# B&R Automation Studio project NAEUL004C00R13L518F00 (part 66)

#### Act_Link.st
```iecst
(** 2021-08-01 **)
ACTION Act_Link:

	//Receive Alive Time
	p_tyParam.tRcvAlive	:= p_tyParam.tSndAlive * 2;

	//Board Depart
	bTransportFinish1 := p_bDSSMEMA1ConvStart AND EDGENEG(p_bPshrConvHvBrd);
	bTransportFinish2 := p_bDSSMEMA2ConvStart AND EDGENEG(p_bPshrConvHvBrd);
	bTransportFinish3 := p_bDSSMEMA3ConvStart AND EDGENEG(p_bPshrConvHvBrd);

	p_bDSHermesTransportFinished1:= bTransportFinish1 OR bTransportFinish2 OR bTransportFinish3;
	//Depart internal SMEMA
	IF EDGEPOS(p_bDSHermesTransportFinished1) THEN// p_bDSHermesTransportFinished1 OR p_bDSHermesTransportFinished2 OR p_bDSHermesTransportFinished3 ) THEN
		memset(ADR(p_bUSHermesARcvBoardInfo),0,SIZEOF(p_bUSHermesARcvBoardInfo));
		IF p_bLinkBrdAvlDataNewBrdAvl1stZ THEN //newly inserted
			//p_tyDSBoardDeparted1.tyData.sBoardId;
			IF NOT(p_bUSHermesARcvBoardInfo) THEN //create new BA
				fHermesGenerateUUID(ADR(tyDsInternalBoardDeparted.tyData.sBoardId) , p_tyDTStructure , pa_usiMacAddr);
				tyDsInternalBoardDeparted.tyData.sBoardIdCreatedBy := p_sMcId;
				tyDsInternalBoardDeparted.tyData.eFailedBoard  := BOOL_TO_USINT(p_bOpsTravLifGdBrdChk)*HermesGoodBoard + BOOL_TO_USINT(NOT(p_bOpsTravLifGdBrdChk))*HermesFailedBoard ;
				tyDsInternalBoardDeparted.tyData.sProductTypeId := p_tyProdRcpCurrRcp1.sRcpNm;
				tyDsInternalBoardDeparted.tyData.sTopBarcode := ''; //from UI
				tyDsInternalBoardDeparted.tyData.sBottomBarcode := ''; //from UI
				tyDsInternalBoardDeparted.tyData.rWidth := DINT_TO_REAL(p_tyProdRcpCurrRcp1.diWidthInUM)/1000;//Rcp
				tyDsInternalBoardDeparted.tyData.rThickness				:= rThickness;
				tyDsInternalBoardDeparted.tyData.rConveyorSpeed			:= rConveyorSpeed;
				tyDsInternalBoardDeparted.tyData.rTopClearanceHeight	:= rTopClearanceHeight;
				tyDsInternalBoardDeparted.tyData.rBottomClearanceHeight	:= rBottomClearanceHeight;
				tyDsInternalBoardDeparted.tyData.rWeight := rWeight;
				tyDsInternalBoardDeparted.tyData.sWorkOrderId := '';
				tyDsInternalBoardDeparted.tyData.sBatchId	:= '';
			ELSE //Take from Send Board Info
				tyDsInternalBoardDeparted.tyData.sBoardId				:= p_tyUSHermesSendBoardInfoAcpt.tyData.sBoardId;
				tyDsInternalBoardDeparted.tyData.sBoardIdCreatedBy 		:= p_tyUSHermesSendBoardInfoAcpt.tyData.sBoardIdCreatedBy;
				tyDsInternalBoardDeparted.tyData.eFailedBoard 			:= p_tyUSHermesSendBoardInfoAcpt.tyData.eFailedBoard;
				tyDsInternalBoardDeparted.tyData.sProductTypeId 		:= p_tyUSHermesSendBoardInfoAcpt.tyData.sProductTypeId;
				tyDsInternalBoardDeparted.tyData.sTopBarcode 			:= p_tyUSHermesSendBoardInfoAcpt.tyData.sTopBarcode;
				tyDsInternalBoardDeparted.tyData.sBottomBarcode 		:= p_tyUSHermesSendBoardInfoAcpt.tyData.sBottomBarcode;
				tyDsInternalBoardDeparted.tyData.rWidth 				:= p_tyUSHermesSendBoardInfoAcpt.tyData.rWidth;//Rcp
				tyDsInternalBoardDeparted.tyData.rThickness				:= p_tyUSHermesSendBoardInfoAcpt.tyData.rThickness;
				tyDsInternalBoardDeparted.tyData.rTopClearanceHeight	:= p_tyUSHermesSendBoardInfoAcpt.tyData.rTopClearanceHeight;
				tyDsInternalBoardDeparted.tyData.rBottomClearanceHeight	:= p_tyUSHermesSendBoardInfoAcpt.tyData.rBottomClearanceHeight;
				tyDsInternalBoardDeparted.tyData.rWeight 				:= p_tyUSHermesSendBoardInfoAcpt.tyData.rWeight;
				tyDsInternalBoardDeparted.tyData.sWorkOrderId 			:= p_tyUSHermesSendBoardInfoAcpt.tyData.sWorkOrderId;
				tyDsInternalBoardDeparted.tyData.sBatchId				:= p_tyUSHermesSendBoardInfoAcpt.tyData.sBatchId;
			END_IF
		ELSE //taken from USHemes
			fbParseBrdAvlExternal.p_XMLTable := ADR(pa_tyLinkXMLTableDataBrdAvl1);
			fbParseBrdAvlExternal.iTotalIdxWrite := p_iLinkXMLTableDataBrdAvlTtlIdx1;
			fbParseBrdAvlExternal;
			tyDsInternalBoardDeparted := fbParseBrdAvlExternal.tyBoardAvailable;
		END_IF
		//differiate
		IF bTransportFinish1 THEN
			sMagazineId := '1';
			iSlotId := DINT_TO_INT(p_diBuffer1Slt);
			p_eBoardTransfer1 := BOOL_TO_USINT(p_bLinkBrdAvlDataNewBrdAvl1stZ)*HermesInserted + BOOL_TO_USINT(NOT(p_bLinkBrdAvlDataNewBrdAvl1stZ))*HermesTransferred;
			p_tyDSBoardDeparted1 := tyDsInternalBoardDeparted;
		ELSIF bTransportFinish2 THEN
			sMagazineId := '2';
			iSlotId	 := DINT_TO_INT(p_diBuffer2Slt);
			p_eBoardTransfer1 := BOOL_TO_USINT(p_bLinkBrdAvlDataNewBrdAvl1stZ)*HermesInserted + BOOL_TO_USINT(NOT(p_bLinkBrdAvlDataNewBrdAvl1stZ))*HermesTransferred;
			p_tyDSBoardDeparted1 := tyDsInternalBoardDeparted;
		ELSIF bTransportFinish3 THEN
			sMagazineId := '3';
			iSlotId := DINT_TO_INT(p_diBuffer3Slt);
			p_eBoardTransfer1 := BOOL_TO_USINT(p_bLinkBrdAvlDataNewBrdAvl1stZ)*HermesInserted + BOOL_TO_USINT(NOT(p_bLinkBrdAvlDataNewBrdAvl1stZ))*HermesTransferred;
			p_tyDSBoardDeparted1 := tyDsInternalBoardDeparted;
		END_IF

	END_IF

//		IF EDGEPOS(p_bDSHermesTransportFinished1) THEN
//			sMagazineId := '1';
//			iSlotId := DINT_TO_INT(p_diBuffer1Slt);
//			p_eBoardTransfer1 := BOOL_TO_USINT(p_bLinkBrdAvlDataNewBrdAvl1stZ)*HermesInserted + BOOL_TO_USINT(NOT(p_bLinkBrdAvlDataNewBrdAvl1stZ))*HermesTransferred;
//			p_tyDSBoardDeparted1 := tyDsInternalBoardDeparted;
//
//		ELSIF EDGEPOS(p_bDSHermesTransportFinished2) THEN
//			sMagazineId := '2';
//			iSlotId	 := DINT_TO_INT(p_diBuffer2Slt);
//			p_eBoardTransfer2 := BOOL_TO_USINT(p_bLinkBrdAvlDataNewBrdAvl1stZ)*HermesInserted + BOOL_TO_USINT(NOT(p_bLinkBrdAvlDataNewBrdAvl1stZ))*HermesTransferred;
//			p_tyDSBoardDeparted2 := tyDsInternalBoardDeparted;
//		ELSIF EDGEPOS(p_bDSHermesTransportFinished3) THEN
//			sMagazineId := '3';
//			iSlotId := DINT_TO_INT(p_diBuffer3Slt);
//			p_eBoardTransfer3 := BOOL_TO_USINT(p_bLinkBrdAvlDataNewBrdAvl1stZ)*HermesInserted + BOOL_TO_USINT(NOT(p_bLinkBrdAvlDataNewBrdAvl1stZ))*HermesTransferred;
//			p_tyDSBoardDeparted3 := tyDsInternalBoardDeparted;
//		END_IF

	//Info Message
	p_sInfoMsg		:= 'Hermes Configuration Received From Supervisory System';

	//Info Message 1
	p_sInfoMsg1     := 'Work Order Info Received From Supervisory System';
	p_sInfoMsg1		:= CONCAT(p_sInfoMsg1 , '$r$n');
	p_sInfoMsg1		:= CONCAT(p_sInfoMsg1 , 'PCB Work Order Info Will Be Overwritten');

	//Info Message 2
//	p_sInfoMsg2     := 'Work Order Info Not Found From Supervisory System';
	p_sInfoMsg2     := 'Work Order Or Data Info Invalid From Supervisory System';
	p_sInfoMsg2		:= CONCAT(p_sInfoMsg2 , '$r$n');
	p_sInfoMsg2  	:= CONCAT(p_sInfoMsg2 , 'Please Try Again');

	//Info Message 3
	p_sInfoMsg3     := 'Query Work Order Not Possible';
	p_sInfoMsg3		:= CONCAT(p_sInfoMsg3 , '$r$n');
	p_sInfoMsg3  	:= CONCAT(p_sInfoMsg3 , 'Please Empty the Machines');
	p_sInfoMsg3		:= CONCAT(p_sInfoMsg3 , '$r$n');
	p_sInfoMsg3  	:= CONCAT(p_sInfoMsg3 , 'and Try Again');

	//Info Message 4
	p_sInfoMsg4     := 'Work Order Info Received From Supervisory System';
	p_sInfoMsg4		:= CONCAT(p_sInfoMsg4 , '$r$n');
	p_sInfoMsg4  	:= CONCAT(p_sInfoMsg4 , 'PCB Work Order Info Will Be Queue for next Batch');

	//Accept WorkOrderId from Supervisory System, adjust accordingly
	//(Loader Machine: Magazine area empty, Lifter area empty)
	//(Destacker Machine: load pcb stack area empty and conveyor empty)
	//Unloader do not accep WO
	p_bAcceptCondition := FALSE;//p_bAllZonesEmpty (*AND p_bUITopUpBrdRdy =FALSE*);

	IF 	p_tyUSBoardAvailableRcv.tyData.sWorkOrderId = '' OR p_tyUSBoardAvailableRcv.tyData.sWorkOrderId <> tySendBypassWorkOrderInfoAcc.tyData.sWorkOrderId OR p_tyUSBoardAvailableRcv.tyData.sBatchId = '' OR  p_tyUSBoardAvailableRcv.tyData.sBatchId <> tySendBypassWorkOrderInfoAcc.tyData.sBatchId OR
		p_tyUSBoardAvailableRcv.tyData.rWidth = 0 OR p_tyUSBoardAvailableRcv.tyData.rWidth <> tySendBypassWorkOrderInfoAcc.tyData.rWidth THEN
		IF p_tyUSBoardAvailableRcv.tyData.sTopBarcode <> '' OR p_tyUSBoardAvailableRcv.tyData.sBottomBarcode <> '' THEN
			sUSBarcode := p_tyUSBoardAvailableRcv.tyData.sTopBarcode;
			bNewIncomingBoard := TRUE;
		ELSIF p_tyUSBoardAvailableRcv.tyAvl.bTopBarcode = FALSE OR p_tyUSBoardAvailableRcv.tyAvl.bBottomBarcode THEN
			sUSBarcode := p_tyUSBoardAvailableRcv.tyData.sBottomBarcode;
			bNewIncomingBoard := TRUE;
		ELSE
			bNewIncomingBoard := FALSE;
		END_IF
	ELSIF p_tyUSBoardForecastRcv.tyAvl.bWorkOrderId OR p_tyUSBoardForecastRcv.tyAvl.bBatchId OR p_tyUSBoardForecastRcv.tyAvl.bWeight THEN

		IF p_tyUSBoardForecastRcv.tyData.sWorkOrderId = '' OR p_tyUSBoardForecastRcv.tyData.sWorkOrderId <> tySendBypassWorkOrderInfoAcc.tyData.sWorkOrderId OR p_tyUSBoardForecastRcv.tyData.sBatchId = '' OR  p_tyUSBoardForecastRcv.tyData.sBatchId <> tySendBypassWorkOrderInfoAcc.tyData.sBatchId OR
			p_tyUSBoardForecastRcv.tyData.rWidth = 0 OR p_tyUSBoardForecastRcv.tyData.rWidth <> tySendBypassWorkOrderInfoAcc.tyData.rWidth THEN

			IF p_tyUSBoardForecastRcv.tyData.sTopBarcode <> '' OR p_tyUSBoardForecastRcv.tyData.sBottomBarcode <> '' THEN

			sUSBarcode := p_tyUSBoardForecastRcv.tyData.sTopBarcode;
			bNewIncomingBoard := TRUE;
			ELSIF p_tyUSBoardForecastRcv.tyAvl.bTopBarcode = FALSE OR p_tyUSBoardForecastRcv.tyAvl.bBottomBarcode THEN
			sUSBarcode := p_tyUSBoardForecastRcv.tyData.sBottomBarcode;
			bNewIncomingBoard := TRUE;
			ELSE
				bNewIncomingBoard := FALSE;
			END_IF
		ELSE
			bNewIncomingBoard := FALSE;
		END_IF
	ELSE
		bNewIncomingBoard := FALSE;
	END_IF

	IF EDGENEG (p_bQueryWorkOrderInfo)  THEN
		IF p_bOpsConvWaitForTopUpBrd THEN
			bManualQueryWO := TRUE;
		ELSIF p_bOpsConvWaitForTopUpBrd = FALSE THEN
			bManualQueryWO := FALSE;
		END_IF
	END_IF

	IF p_bOpsConvWaitForTopUpBrd = FALSE THEN
		bManualQueryWO := FALSE;
	END_IF

	IF diReqLoaderWidthInUM = 0 THEN                           //Load Data during bootup
		diReqLoaderWidthInUM := REAL_TO_DINT(tySendWorkOrderInfoAcc.tyData.rWidth * 1000);
	END_IF

	IF EDGENEG (p_bLinkStartupRun) THEN
		sWorkOrderId := tySendWorkOrderInfoNewAcc.tyData.sWorkOrderId;
	END_IF

	//	phase 2
//	bChangeOverLifter := lifterEmpty + no UBA + waitTimeOut;
//	bChangeOverLoader := lifterEmpty + UBA + waitTimeOut;
//	IF  p_bAcceptConditionLifter  THEN
//		tySendWorkOrderInfoAccPublish := tySendWorkOrderInfoAcc;
//	ELSIF  p_bAcceptConditionLoader  THEN
//		tySendWorkOrderInfoAccPublish := tySendWorkOrderInfoAcc;
//	END_IF
END_ACTION
```

#### Act_Main.st
```iecst
(** 2021-08-01 **)
ACTION Act_Main:

	IF eStatOld <> eStat THEN
		fbFileOldDel1(bEn := FALSE);
		fbFileRead1(bEn := FALSE);
		fbFileWrite1(bEn := FALSE);
		bFileNotFound	:= FALSE;
		sStatTxt	:= a_sStatText[eStat];

		eStatOld	:= eStat;

		eStatus		:= Busy;
	END_IF

	//Main
	CASE eStat OF

		HermesActIdle:
			eStatus	:= Idle;

		HermesActBGStartRun:
			IF eStatus = Idle OR eStatus = Busy THEN

				bRun	:= TRUE;
				bStop	:= FALSE;
				eStatus	:= Done;

			END_IF

		HermesActBGStopRun:
			IF eStatus = Idle OR eStatus = Busy THEN

				bStop	:= TRUE;
				eStatus	:= Done;

			END_IF

		HermesActDeleteOldLog:
			IF eStatus = Idle OR eStatus = Busy THEN

				eStatus	:= Busy;

				fbFileOldDel1.dtDTNow	:= p_dtCurrDT;
				fbFileOldDel1(bEn := TRUE);
				IF fbFileOldDel1.udiStatus = 0 THEN
					eStatus	:= Done;
				ELSIF fbFileOldDel1.udiStatus < 65534 THEN
					eStatus		:= Error;

					IF fbFileOldDel1.udiStatus = 1910 THEN
						udiStatus	:= 10111;	//Get Directory Info Error While Deleting Old Log
					ELSIF fbFileOldDel1.udiStatus = 1911 THEN
						udiStatus	:= 10112;	//Directory Read Error While Deleting Old Log
					ELSIF fbFileOldDel1.udiStatus = 1912 THEN
						udiStatus	:= 10113;	//File Delete Error While Deleting Old Log
					ELSE
						udiStatus	:= fbFileOldDel1.udiStatus;
					END_IF
				END_IF

			END_IF

		HermesActReadRetain:
			IF eStatus = Idle OR eStatus = Busy THEN

				eStatus	:= Busy;

				fbFileRead1.p_Dest	:= p_udiRetainDataAddr;
				fbFileRead1.udiLen	:= p_udiRetainDataLen;
				fbFileRead1(bEn := TRUE);

				IF fbFileRead1.udiStatus = 0 THEN
					eStatus	:= Done;
				ELSIF fbFileRead1.udiStatus < 65534 THEN
					eStatus	:= Error;

					IF fbFileRead1.udiStatus = 1900 THEN
						udiStatus	:= 10114;	//File Open Error While Reading Retain File
					ELSIF fbFileRead1.udiStatus = 1902 THEN
						udiStatus	:= 10115;	//File Read Error While Reading Retain File
					ELSIF fbFileRead1.udiStatus = 1904 THEN
						udiStatus	:= 10116;	//File Close Error While Reading Retain File
					ELSIF fbFileRead1.udiStatus = 1915 THEN
						eStatus			:= Done;
						bFileNotFound	:= TRUE;
					ELSE
						udiStatus	:= fbFileRead1.udiStatus;
					END_IF
				END_IF

			END_IF

		HermesActWriteRetain:
			IF eStatus = Idle OR eStatus = Busy THEN

				eStatus	:= Busy;

				fbFileWrite1.p_Src	:= p_udiRetainDataAddr;
				fbFileWrite1.udiLen	:= p_udiRetainDataLen;
				fbFileWrite1(bEn := TRUE);

				IF fbFileWrite1.udiStatus = 0 THEN
					eStatus	:= Done;
				ELSIF fbFileWrite1.udiStatus < 65534 THEN
					eStatus	:= Error;

					IF fbFileWrite1.udiStatus = 1900 THEN
						udiStatus	:= 10117;	//File Open Error While Writing Retain File
					ELSIF fbFileWrite1.udiStatus = 1901 THEN
						udiStatus	:= 10118;	//File Create Error While Writing Retain File
					ELSIF fbFileWrite1.udiStatus = 1903 THEN
						udiStatus	:= 10119;	//File Write Error While Writing Retain File
					ELSIF fbFileWrite1.udiStatus = 1904 THEN
						udiStatus	:= 10120;	//File Close Error While Writing Retain File
					ELSIF fbFileWrite1.udiStatus = 1914 THEN
						udiStatus	:= 10121;	//Directory Does Not Exist While Writing Retain File
					ELSE
						udiStatus	:= fbFileWrite1.udiStatus;
					END_IF
				END_IF

			END_IF

		HermesActReadRetainSendWO1:
			IF eStatus = Idle OR eStatus = Busy THEN

				eStatus	:= Busy;

				fbFileRead2.p_Dest	:= p_udiLoaderRetainDataAddr0;
				fbFileRead2.udiLen	:= p_udiLoaderRetainDataLen0;
				fbFileRead2(bEn := TRUE);

				IF fbFileRead2.udiStatus = 0 THEN
					eStatus	:= Done;
				ELSIF fbFileRead2.udiStatus < 65534 THEN
					eStatus	:= Error;

					IF fbFileRead2.udiStatus = 1900 THEN
						udiStatus	:= 10200;	//File Open Error While Reading Retain File
					ELSIF fbFileRead2.udiStatus = 1902 THEN
						udiStatus	:= 10201;	//File Read Error While Reading Retain File
					ELSIF fbFileRead2.udiStatus = 1904 THEN
						udiStatus	:= 10202;	//File Close Error While Reading Retain File
					ELSIF fbFileRead2.udiStatus = 1915 THEN
						eStatus			:= Done;
						bFileNotFound	:= TRUE;
					ELSE
						udiStatus	:= fbFileRead2.udiStatus;
					END_IF
				END_IF

			END_IF

		HermesActWriteRetainSendWO1:
			IF eStatus = Idle OR eStatus = Busy THEN

				eStatus	:= Busy;

				fbFileWrite2.p_Src	:= p_udiLoaderRetainDataAddr0;
				fbFileWrite2.udiLen	:= p_udiLoaderRetainDataLen0;
				fbFileWrite2(bEn := TRUE);

				IF fbFileWrite2.udiStatus = 0 THEN
					eStatus	:= Done;
				ELSIF fbFileWrite2.udiStatus < 65534 THEN
					eStatus	:= Error;

					IF fbFileWrite2.udiStatus = 1900 THEN
						udiStatus	:= 10203;	//File Open Error While Writing Retain File
					ELSIF fbFileWrite2.udiStatus = 1901 THEN
						udiStatus	:= 10204;	//File Create Error While Writing Retain File
					ELSIF fbFileWrite2.udiStatus = 1903 THEN
						udiStatus	:= 10205;	//File Write Error While Writing Retain File
					ELSIF fbFileWrite2.udiStatus = 1904 THEN
						udiStatus	:= 10206;	//File Close Error While Writing Retain File
					ELSIF fbFileWrite2.udiStatus = 1914 THEN
						udiStatus	:= 10207;	//Directory Does Not Exist While Writing Retain File
					ELSE
						udiStatus	:= fbFileWrite2.udiStatus;
					END_IF
				END_IF

			END_IF

		HermesActReadRetainSendWO2:
			IF eStatus = Idle OR eStatus = Busy THEN

				eStatus	:= Busy;

				fbFileRead3.p_Dest	:= p_udiLoaderRetainDataAddr1;
				fbFileRead3.udiLen	:= p_udiLoaderRetainDataLen1;
				fbFileRead3(bEn := TRUE);

				IF fbFileRead3.udiStatus = 0 THEN
					eStatus	:= Done;
				ELSIF fbFileRead3.udiStatus < 65534 THEN
					eStatus	:= Error;

					IF fbFileRead3.udiStatus = 1900 THEN
						udiStatus	:= 10208;	//File Open Error While Reading Retain File
					ELSIF fbFileRead3.udiStatus = 1902 THEN
						udiStatus	:= 10209;	//File Read Error While Reading Retain File
					ELSIF fbFileRead3.udiStatus = 1904 THEN
						udiStatus	:= 10210;	//File Close Error While Reading Retain File
					ELSIF fbFileRead3.udiStatus = 1915 THEN
						eStatus			:= Done;
						bFileNotFound	:= TRUE;
					ELSE
						udiStatus	:= fbFileRead3.udiStatus;
					END_IF
				END_IF

			END_IF

		HermesActWriteRetainSendWO2:
			IF eStatus = Idle OR eStatus = Busy THEN

				eStatus	:= Busy;

				fbFileWrite3.p_Src	:= p_udiLoaderRetainDataAddr1;
				fbFileWrite3.udiLen	:= p_udiLoaderRetainDataLen1;
				fbFileWrite3(bEn := TRUE);

				IF fbFileWrite3.udiStatus = 0 THEN
					eStatus	:= Done;
				ELSIF fbFileWrite3.udiStatus < 65534 THEN
					eStatus	:= Error;

					IF fbFileWrite3.udiStatus = 1900 THEN
						udiStatus	:= 10211;	//File Open Error While Writing Retain File
					ELSIF fbFileWrite3.udiStatus = 1901 THEN
						udiStatus	:= 10212;	//File Create Error While Writing Retain File
					ELSIF fbFileWrite3.udiStatus = 1903 THEN
						udiStatus	:= 10213;	//File Write Error While Writing Retain File
					ELSIF fbFileWrite3.udiStatus = 1904 THEN
						udiStatus	:= 10214;	//File Close Error While Writing Retain File
					ELSIF fbFileWrite3.udiStatus = 1914 THEN
						udiStatus	:= 10215;	//Directory Does Not Exist While Writing Retain File
					ELSE
						udiStatus	:= fbFileWrite3.udiStatus;
					END_IF
				END_IF

			END_IF

		HermesActReadRetainSendWO3:
			IF eStatus = Idle OR eStatus = Busy THEN

				eStatus	:= Busy;

				fbFileRead4.p_Dest	:= p_udiBypassRetainDataAddr0;
				fbFileRead4.udiLen	:= p_udiBypassRetainDataLen0;
				fbFileRead4(bEn := TRUE);

				IF fbFileRead4.udiStatus = 0 THEN
					eStatus	:= Done;
				ELSIF fbFileRead4.udiStatus < 65534 THEN
					eStatus	:= Error;

					IF fbFileRead4.udiStatus = 1900 THEN
						udiStatus	:= 10216;	//File Open Error While Reading Retain File
					ELSIF fbFileRead4.udiStatus = 1902 THEN
						udiStatus	:= 10217;	//File Read Error While Reading Retain File
					ELSIF fbFileRead4.udiStatus = 1904 THEN
						udiStatus	:= 10218;	//File Close Error While Reading Retain File
					ELSIF fbFileRead4.udiStatus = 1915 THEN
						eStatus			:= Done;
						bFileNotFound	:= TRUE;
					ELSE
						udiStatus	:= fbFileRead4.udiStatus;
					END_IF
				END_IF

			END_IF

		HermesActWriteRetainSendWO3:
			IF eStatus = Idle OR eStatus = Busy THEN

				eStatus	:= Busy;

				fbFileWrite4.p_Src	:= p_udiBypassRetainDataAddr0;
				fbFileWrite4.udiLen	:= p_udiBypassRetainDataLen0;
				fbFileWrite4(bEn := TRUE);

				IF fbFileWrite4.udiStatus = 0 THEN
					eStatus	:= Done;
				ELSIF fbFileWrite4.udiStatus < 65534 THEN
					eStatus	:= Error;

					IF fbFileWrite4.udiStatus = 1900 THEN
						udiStatus	:= 10219;	//File Open Error While Writing Retain File
					ELSIF fbFileWrite4.udiStatus = 1901 THEN
						udiStatus	:= 10220;	//File Create Error While Writing Retain File
					ELSIF fbFileWrite4.udiStatus = 1903 THEN
						udiStatus	:= 10221;	//File Write Error While Writing Retain File
					ELSIF fbFileWrite4.udiStatus = 1904 THEN
						udiStatus	:= 10222;	//File Close Error While Writing Retain File
					ELSIF fbFileWrite4.udiStatus = 1914 THEN
						udiStatus	:= 10223;	//Directory Does Not Exist While Writing Retain File
					ELSE
						udiStatus	:= fbFileWrite4.udiStatus;
					END_IF
				END_IF

			END_IF

		ELSE
			IF eStatus = Idle OR eStatus = Busy THEN
				eStatus	:= Done;
			END_IF

	END_CASE

END_ACTION
```

#### Init.st
```iecst
(** 2021-08-01 **)
PROGRAM _INIT

	(* Always Change If Project Change *)

	//Pass Address To Global Address For External Use
	//Action, State & Status
	p_SvyHermesStat	    	:= ADR(eStat);
	p_SvyHermesStatus   	:= ADR(eMainStatus);
	p_SvyHermesStatTxt    	:= ADR(sStatTxt);
	p_SvyHermesAct	    	:= ADR(eHermesAct);
	p_SvyHermesMcParamAct	:= ADR(eMcParamAct);

	//Alarm
	p_SvyHermesAlmData	    := ADR(tyAlmData);
	p_SvyHermesAlmData1	    := ADR(tyAlmData1);
	p_SvyHermesAlmData2	    := ADR(tyAlmData2);
	p_SvyHermesAlmData3	    := ADR(tyAlmData3);
    p_SvyHermesAlmData4	    := ADR(tyAlmData4);
	p_SvyHermesInfoData	    := ADR(tyInfoData);
	p_SvyHermesInfoData1	:= ADR(tyInfoData1);
	p_SvyHermesInfoData2	:= ADR(tyInfoData2);
	p_SvyHermesInfoData3	:= ADR(tyInfoData3);
	p_SvyHermesInfoData4	:= ADR(tyInfoData4);

	//Output
	p_SvyHermesConnected			:= ADR(bConnected);
	p_SvyHermesHandshakeDone		:= ADR(bHandshakeDone);
	p_SvyHermesInternalSnd		    := ADR(sInternalSnd);
	p_SvyHermesFileNotFound			:= ADR(bFileNotFound);
	p_SvyHermesSetConfiguration	    := ADR(tySetConfigurationModified);
	p_SvyHermesWriteConfig	        := ADR(bWriteConfig);
	p_SvyHermesUpdateUIData	        := ADR(bUpdateUIData);
	p_SvyHermesWorkOrderId          := ADR(sWorkOrderId); //WorkOrderId from Supervisory System
	p_SvyHermesBatchId              := ADR(sBatchId); //BatchId from Supervisory System

	//Data
	p_SvyHermesFoundIndexUS1              := ADR(bFoundIndexUS1);
	p_SvyHermesFoundIndexUS2              := ADR(bFoundIndexUS2);
	p_SvyHermesFoundIndexUS3              := ADR(bFoundIndexUS3);
	p_SvyHermesFoundIndexUS4              := ADR(bFoundIndexUS4);
	p_SvyHermesFoundIndexDS1              := ADR(bFoundIndexDS1);
	p_SvyHermesFoundIndexDS2              := ADR(bFoundIndexDS2);
	p_SvyHermesFoundIndexDS3              := ADR(bFoundIndexDS3);
	p_SvyHermesFoundIndexDS4              := ADR(bFoundIndexDS4);
	p_SvyHermesIndexUS1                   := ADR(udiFoundIndexUS1);
	p_SvyHermesIndexUS2                   := ADR(udiFoundIndexUS2);
	p_SvyHermesIndexUS3                   := ADR(udiFoundIndexUS3);
	p_SvyHermesIndexUS4                   := ADR(udiFoundIndexUS4);
	p_SvyHermesIndexDS1                   := ADR(udiFoundIndexDS1);
	p_SvyHermesIndexDS2                   := ADR(udiFoundIndexDS2);
	p_SvyHermesIndexDS3                   := ADR(udiFoundIndexDS3);
	p_SvyHermesIndexDS4                   := ADR(udiFoundIndexDS4);
	p_RcvBoardInfoOk                      := ADR(bRcvBoardInfoOk);

	//Publish  this to USHermes

	//phase 1
	p_SvyHermesSendWorkOrderData       := ADR(tySendWorkOrderInfoNewAcc);
	p_SvyHermesBypassSendWOData        := ADR (tySendBypassWorkOrderInfoAcc);
	p_ReplyWorkOrderInfo               := ADR(bReplyWorkOrderInfo);
	p_SendBoardForecast                := ADR (bSendBoardForecast);
	p_ClearWorkOrder                   := ADR (bClearWorkOrder);
    p_NewIncomingBoard                 := ADR (bNewIncomingBoard);
	p_QueryBypassWorkOrder             := ADR (bQueryBypassWorkOrder);
	p_ReplyBypassWorkOrderInfo         := ADR (bReplyBypassWorkOrderInfo);
	p_ReqLoaderWidthInUM               := ADR  (diReqLoaderWidthInUM);
	p_RcvWorkOrderInfo1                := ADR  (bRcvWorkOrderInfo1);

	//phase 2
	//tySendWorkOrderInfoAccPublish
	(* Always Change If Project Change *)

END_PROGRAM
```

### LCS.typ - Change By Project
```iecst
(*2019-07-10*)
(**)
(*Action*)

TYPE
	eLCSAction :
		(
		LCSActIdle := 0,
		LCSActAddProd := 1,
		LCSActAddMultiProd := 2,
		LCSActEditProd := 3,
		LCSActEditMultiProd := 4,
		LCSActOverWriteProd := 5,
		LCSActOverWriteMultiProd := 6,
		LCSActDelProd := 7,
		LCSActDelMultiProd := 8,
		LCSActRunProd := 9,
		LCSActUploadProd := 10,
		LCSActUploadMultiProd := 11,
		LCSActOverWriteMag := 12,
		LCSActDelMag := 13,
		LCSActUploadMag := 14
		);
END_TYPE

(**)
(*Data*)

TYPE
	eLCSOpsStatus :
		(
		LCSOpsStatusAuto,
		LCSOpsStatusManual,
		LCSOpsStatusStop,
		LCSOpsStatusError,
		LCSOpsStatusWarning
		);
	tyLCSTagNm : 	STRUCT
		eAct : eLCSAction;
		eStat : eLCSAction;
		udiStatus : UDINT;
		sErrMsg : STRING[200];
		iIdxAct : INT;
		iIdxStat : INT;
		tyProdRcpInfo : tyProdRcpParam;
		tyCurrProdRcpParam : tyProdRcpParam;
		sCurrRcpNm : STRING[30];
		rCurrWidth : REAL;
		eCurrOpsStatus : eLCSOpsStatus;
		usiBrdStatus : USINT;
		usiMode : USINT;
		iTopToBtm : INT;
		sLastModified : STRING[80];
		bMngRcpEn : BOOL;
		bLiveData : BOOL;
		bLFEn : BOOL;
		sMcAlmMsg : ARRAY[1..c_udiAlarmCurrMax]OF STRING[255];
		bSectionLeaderEn : BOOL;
		bBlkUS : BOOL;
		bBlkDS : BOOL;
		tyMagRcpInfo : tyMagRcpParam;
		tyCurrMagRcpParam : tyMagRcpParam;
		sCurrMagRcpNm : STRING[15];
	END_STRUCT;
END_TYPE
```

### LCS.var - Change By Project
```iecst
(*2019-04-24*)
(**)
(*Action & State & Status*)
(**)
(*Alarm*)
(**)
(*Output*)
VAR
	p_LCS_LCSMngRcp_LCSAct : UDINT;
	p_LCS_LCSMngRcp_LCSIdxAct : UDINT;
	p_LCS_LCSMngRcp_LCSIdxStat : UDINT;
	p_LCS_LCSMngRcp_LCSProdRcpInfo : UDINT;
	p_LCS_LCSLF_LCSAct : UDINT;
	p_LCS_LCSLF_LCSProdRcpInfo : UDINT;
	p_LCSChkLmtOK : UDINT;
	p_LCSChkLmtNG : UDINT;
	p_LCS_LCSMngRcp_LCSMagRcpInfo : UDINT;
	p_LCSChkMagLmtOK : UDINT;
	p_LCSChkMagLmtNG : UDINT;
	p_LCSSectionLeaderEn : UDINT;
END_VAR
```

### Program Logical/LCS/LCS (IEC, version 1.00.0) - 1.00.0 - NtRecipe v5.00.0 , NtFileIO v5.00.0

#### Init.st - Change By Project
```iecst
(** 2019-04-24 **)
PROGRAM _INIT

	(* Always Change If Project Change *)

	//Pass Address To Global Address For External Use
	//Action, State & Status

	//Alarm

	//Output
	p_LCS_LCSMngRcp_LCSAct			:= ADR(eLCSMngRcp_LCSAct);
	p_LCS_LCSMngRcp_LCSIdxAct		:= ADR(iLCSMngRcp_LCSIdxAct);
	p_LCS_LCSMngRcp_LCSIdxStat		:= ADR(iLCSMngRcp_LCSIdxStat);
	p_LCS_LCSMngRcp_LCSProdRcpInfo	:= ADR(tyLCSMngRcp_LCSProdRcpInfo);
	p_LCS_LCSLF_LCSAct				:= ADR(eLCSLF_LCSAct);
	p_LCS_LCSLF_LCSProdRcpInfo		:= ADR(tyLCSLF_LCSProdRcpInfo);
	p_LCSChkLmtOK					:= ADR(bChkLmtOK);
	p_LCSChkLmtNG					:= ADR(bChkLmtNG);

	p_LCS_LCSMngRcp_LCSMagRcpInfo 	:= ADR(tyLCSMngRcp_LCSMagRcpInfo);
	p_LCSChkMagLmtOK					:= ADR(bChkMagLmtOk);
	p_LCSChkMagLmtNG					:= ADR(bChkMagLmtNG);
	p_LCSSectionLeaderEn 				:= ADR(tyTagNm.bSectionLeaderEn);
	(* Always Change If Project Change *)

END_PROGRAM
```

#### Act_InitGlobal.st - Change By Project
```iecst
(** 2019-06-12 **)
ACTION Act_InitGlobal:

	(* Always Change If Project Change *)

	//Pass Data To Link
	p_bLinkStartupRun ACCESS p_StartupRun;
	p_bLinkNtParamProjLaneBPrep ACCESS p_NtParamProjLaneBPrep;
	p_bLinkNtParamLCSLFPrep ACCESS p_NtParamLCSLFPrep;
	p_bLinkNtParamLCSManageRcpPrep ACCESS p_NtParamLCSManageRcpPrep;
	p_bLinkNtParamLCSReqRcpPrep ACCESS p_NtParamLCSReqRcpPrep;
	p_bLinkNtParamLCSLiveDatPrep ACCESS p_NtParamLCSLiveDatPrep;
	p_bLinkMcParamLCSLFEn ACCESS p_McParamLCSLFEn;
	p_bLinkMcParamLCSManageRcpEn ACCESS p_McParamLCSManageRcpEn;
	p_bLinkMcParamLCSReqRcpEn ACCESS p_McParamLCSReqRcpEn;
	p_bLinkMcParamLCSLiveDatEn ACCESS p_McParamLCSLiveDatEn;
	p_tyLinkMcParamMagParamSelected ACCESS p_MagRcpCurrRcp;
	p_bLinkPshrConvHvBrd ACCESS p_PshrConvHvBrd;
	p_eLinkNtParamProjMag ACCESS p_NtParamProjMag;
	p_bLinkBffr1MagRemoved ACCESS p_Buffer1MagRemoved;
	p_bLinkBffr2MagRemoved ACCESS p_Buffer2MagRemoved;
	p_bLinkBffr3MagRemoved ACCESS p_Buffer3MagRemoved;
	p_tyLinkAlarmCurrList ACCESS p_AlarmCurrList;

	//Pass Data To Internal Use
	p_eLCSMngRcp_PLCStat ACCESS p_LCSMngRcpStat;
	p_udiLCSMngRcp_PLCStatus ACCESS p_LCSMngRcp_PLCStatus;
	p_iLCSMngRcp_PLCIdxAct ACCESS p_LCSMngRcp_PLCIdxAct;
	p_iLCSMngRcp_PLCIdxStat ACCESS p_LCSMngRcp_PLCIdxStat;
	p_tyLCSMngRcp_PLCProdRcpInfo ACCESS p_LCSMngRcp_PLCProdRcpInfo;
	p_eLCSLF_PLCStat ACCESS p_LCSLFStat;
	p_udiLCSLF_PLCStatus ACCESS p_LCSLF_PLCStatus;
	p_bLCSMngRcpChkLmt ACCESS p_LCSMngRcpChkLmt;
	p_bLCSLFChkLmt ACCESS p_LCSLFChkLmt;
	p_bOpsRun ACCESS p_OpsRun;
	p_bError ACCESS p_AlarmErr;
	p_bWarning ACCESS p_AlarmWarning;
	p_bInfo ACCESS p_AlarmInfo;
	p_bUIManual ACCESS p_UIUIMnlMod;
	p_tyProdRcpCurrRcp ACCESS p_Follower2UpdtProdRcp;	//Assign With Conveyor Last Zone (Live Data Update)
	p_tyNtParamCurr ACCESS p_NtParamCurr;
	p_sProgNm ACCESS p_NtParamLCSProgNm;
	p_bNtSettingsLoadDone ACCESS p_StartupNtSettingsLoadDone;
		(* Always Change If Project Change *)
	p_tyMagRcpCurrRcp ACCESS p_MagRcpCurrRcp; //LCS Added
	p_tyLCSMngRcp_PLCMagRcpInfo ACCESS p_LCSMngRcp_PLCMagRcpInfo;
	p_bLCSMngMagRcpChkLmt ACCESS p_LCSMngMagRcpChkLmt;

END_ACTION
```

#### InputRef_Link.var - Change By Project
```iecst
(*2019-04-24*)
(**)
VAR
	p_bLinkStartupRun : REFERENCE TO BOOL;
	p_bLinkNtParamProjLaneBPrep : REFERENCE TO BOOL;
	p_bLinkNtParamLCSLFPrep : REFERENCE TO BOOL;
	p_bLinkNtParamLCSManageRcpPrep : REFERENCE TO BOOL;
	p_bLinkNtParamLCSReqRcpPrep : REFERENCE TO BOOL;
	p_bLinkNtParamLCSLiveDatPrep : REFERENCE TO BOOL;
	p_bLinkMcParamLCSLFEn : REFERENCE TO BOOL;
	p_bLinkMcParamLCSManageRcpEn : REFERENCE TO BOOL;
	p_bLinkMcParamLCSReqRcpEn : REFERENCE TO BOOL;
	p_bLinkMcParamLCSLiveDatEn : REFERENCE TO BOOL;
	p_tyLinkMcParamMagParamSelected : REFERENCE TO tyMagRcpParam;
END_VAR
(**)
VAR
	p_bLinkPshrConvHvBrd : REFERENCE TO BOOL;
	p_eLinkNtParamProjMag : REFERENCE TO eULMag;
	p_bLinkBffr1MagRemoved : REFERENCE TO BOOL;
	p_bLinkBffr2MagRemoved : REFERENCE TO BOOL;
	p_bLinkBffr3MagRemoved : REFERENCE TO BOOL;
	p_tyLinkAlarmCurrList : REFERENCE TO ARRAY[1..c_udiAlarmCurrMax] OF tyAlarmCurr;
END_VAR
```

#### Act_Link.st - Change By Project
```iecst
(** 2019-07-15 **)
ACTION Act_Link:

	//Check Limit
	IF p_bLCSMngRcpChkLmt OR p_bLCSLFChkLmt THEN

		IF tyTagNm.tyProdRcpInfo.sRcpNm = '' THEN

			bChkLmtOK	:= FALSE;
			bChkLmtNG	:= TRUE;
			sAddMsg		:= 'Recipe Name Empty ';

		ELSIF tyTagNm.tyProdRcpInfo.diWidthInUM < p_tyNtParamCurr.tyProdRcpWidth.diMin THEN

			bChkLmtOK	:= FALSE;
			bChkLmtNG	:= TRUE;
			sAddMsg		:= 'Width Lower Limit ';

		ELSIF tyTagNm.tyProdRcpInfo.diWidthInUM > p_tyNtParamCurr.tyProdRcpWidth.diMax THEN

			bChkLmtOK	:= FALSE;
			bChkLmtNG	:= TRUE;
			sAddMsg		:= 'Width Upper Limit ';

		ELSIF NOT p_bLinkNtParamProjLaneBPrep AND (tyTagNm.tyProdRcpInfo.usiMcMod < DINT_TO_USINT(p_tyNtParamCurr.tyProdRcpMcModA.diMin)) THEN

			bChkLmtOK	:= FALSE;
			bChkLmtNG	:= TRUE;
			sAddMsg		:= 'Machine Mode Lower Limit ';

		ELSIF NOT p_bLinkNtParamProjLaneBPrep AND (tyTagNm.tyProdRcpInfo.usiMcMod > DINT_TO_USINT(p_tyNtParamCurr.tyProdRcpMcModA.diMax)) THEN

			bChkLmtOK	:= FALSE;
			bChkLmtNG	:= TRUE;
			sAddMsg		:= 'Machine Mode Upper Limit ';

		ELSIF p_bLinkNtParamProjLaneBPrep AND (tyTagNm.tyProdRcpInfo.usiMcMod < DINT_TO_USINT(p_tyNtParamCurr.tyProdRcpMcModAB.diMin)) THEN

			bChkLmtOK	:= FALSE;
			bChkLmtNG	:= TRUE;
			sAddMsg		:= 'Machine Mode Lower Limit ';

		ELSIF p_bLinkNtParamProjLaneBPrep AND (tyTagNm.tyProdRcpInfo.usiMcMod > DINT_TO_USINT(p_tyNtParamCurr.tyProdRcpMcModAB.diMax)) THEN

			bChkLmtOK	:= FALSE;
			bChkLmtNG	:= TRUE;
			sAddMsg		:= 'Machine Mode Upper Limit ';

		ELSIF tyTagNm.tyProdRcpInfo.diMaxSltValue < tyTagNm.tyProdRcpInfo.diMinSltValue THEN

			bChkLmtOK	:= FALSE;
			bChkLmtNG	:= TRUE;
			sAddMsg		:= 'Max Slot Lower Limit ';

		ELSIF tyTagNm.tyProdRcpInfo.diMaxSltValue > p_tyLinkMcParamMagParamSelected.diTtlSlt THEN

			bChkLmtOK	:= FALSE;
			bChkLmtNG	:= TRUE;
			sAddMsg		:= 'Max Slot Upper Limit ';

		ELSIF tyTagNm.tyProdRcpInfo.diMinSltValue < p_tyNtParamCurr.diProjMagMinSlt THEN

			bChkLmtOK	:= FALSE;
			bChkLmtNG	:= TRUE;
			sAddMsg		:= 'Min Slot Lower Limit ';

		ELSIF tyTagNm.tyProdRcpInfo.diMinSltValue > tyTagNm.tyProdRcpInfo.diMaxSltValue THEN

			bChkLmtOK	:= FALSE;
			bChkLmtNG	:= TRUE;
			sAddMsg		:= 'Min Slot Upper Limit ';

		ELSIF tyTagNm.tyProdRcpInfo.diPitch < p_tyNtParamCurr.tyProdRcpPitch.diMin THEN

			bChkLmtOK	:= FALSE;
			bChkLmtNG	:= TRUE;
			sAddMsg		:= 'Pitch Lower Limit ';

		ELSIF tyTagNm.tyProdRcpInfo.diPitch > (tyTagNm.tyProdRcpInfo.diMaxSltValue - tyTagNm.tyProdRcpInfo.diMinSltValue + 1) THEN

			bChkLmtOK	:= FALSE;
			bChkLmtNG	:= TRUE;
			sAddMsg		:= 'Pitch Upper Limit ';

		ELSIF tyTagNm.tyProdRcpInfo.diMinReqFreeBffr < p_tyNtParamCurr.tyProdRcpOvenMinReqFreeBffr.diMin THEN

			bChkLmtOK	:= FALSE;
			bChkLmtNG	:= TRUE;
			sAddMsg		:= 'Minimum Required Free Buffer Lower Limit ';

		ELSIF tyTagNm.tyProdRcpInfo.diMinReqFreeBffr > p_tyNtParamCurr.tyProdRcpOvenMinReqFreeBffr.diMax THEN

			bChkLmtOK	:= FALSE;
			bChkLmtNG	:= TRUE;
			sAddMsg		:= 'Minimum Required Free Buffer Upper Limit ';

		ELSE

			bChkLmtOK	:= TRUE;
			bChkLmtNG	:= FALSE;
			sAddMsg		:= '';

		END_IF

	ELSE

		bChkLmtOK	:= FALSE;
		bChkLmtNG	:= FALSE;

	END_IF

	IF p_bLCSMngMagRcpChkLmt THEN
		IF tyTagNm.tyMagRcpInfo.sRcpNm = '' THEN

			bChkMagLmtOk	:= FALSE;
			bChkMagLmtNG	:= TRUE;
			sAddMsg		:= 'Magazine Recipe Name Empty ';
		ELSIF tyTagNm.tyMagRcpInfo.diMag1Slt1PosInUM < p_tyNtParamCurr.tyUILifterTargetPos.diMin OR
			tyTagNm.tyMagRcpInfo.diMag2Slt1PosInUM < p_tyNtParamCurr.tyUILifterTargetPos.diMin OR
			tyTagNm.tyMagRcpInfo.diMag3Slt1PosInUM < p_tyNtParamCurr.tyUILifterTargetPos.diMin
			THEN

			bChkMagLmtOk	:= FALSE;
			bChkMagLmtNG	:= TRUE;
			sAddMsg		:= 'Magazine Slot 1 Lower Limit ';

		ELSIF tyTagNm.tyMagRcpInfo.diMag1Slt1PosInUM > p_tyNtParamCurr.tyUILifterTargetPos.diMax OR
			tyTagNm.tyMagRcpInfo.diMag2Slt1PosInUM > p_tyNtParamCurr.tyUILifterTargetPos.diMax OR
			tyTagNm.tyMagRcpInfo.diMag3Slt1PosInUM > p_tyNtParamCurr.tyUILifterTargetPos.diMax
			THEN

			bChkMagLmtOk	:= FALSE;
			bChkMagLmtNG	:= TRUE;
			sAddMsg		:= 'Magazine Slot 1 Upper Limit ';

		ELSIF tyTagNm.tyMagRcpInfo.diSltToSltInUM < p_tyNtParamCurr.tyUISltToSltDist.diMin THEN
			bChkMagLmtOk	:= FALSE;
			bChkMagLmtNG	:= TRUE;
			sAddMsg		:= 'Slot to Slot Lower Limit ';

		ELSIF tyTagNm.tyMagRcpInfo.diSltToSltInUM > p_tyNtParamCurr.tyUISltToSltDist.diMax THEN
			bChkMagLmtOk	:= FALSE;
			bChkMagLmtNG	:= TRUE;
			sAddMsg		:= 'Slot to Slot Upper Limit ';

		ELSIF tyTagNm.tyMagRcpInfo.diTtlSlt < p_tyNtParamCurr.diProjMagMinSlt THEN
			bChkMagLmtOk	:= FALSE;
			bChkMagLmtNG	:= TRUE;
			sAddMsg		:= 'Total Slot Lower Limit ';

		ELSIF tyTagNm.tyMagRcpInfo.diTtlSlt > p_tyNtParamCurr.diProjMagMaxSlt THEN
			bChkMagLmtOk	:= FALSE;
			bChkMagLmtNG	:= TRUE;
			sAddMsg		:= 'Total Slot Upper Limit ';
		ELSIF tyTagNm.tyMagRcpInfo.usiMagModel < 0 THEN
			bChkMagLmtOk	:= FALSE;
			bChkMagLmtNG	:= TRUE;
			sAddMsg		:= 'Magazine Model Lower Limit ';
		ELSIF tyTagNm.tyMagRcpInfo.usiMagModel > 2 THEN
			bChkMagLmtOk	:= FALSE;
			bChkMagLmtNG	:= TRUE;
			sAddMsg		:= 'Magazine Model Upper Limit ';
		ELSIF tyTagNm.tyMagRcpInfo.diMagMaxBrdWidth < p_tyNtParamCurr.tyProdRcpWidth.diMin THEN
			bChkMagLmtOk	:= FALSE;
			bChkMagLmtNG	:= TRUE;
			sAddMsg		:= 'Maximum Board Width Upper Limit ';
		ELSIF tyTagNm.tyMagRcpInfo.diMagMaxBrdWidth > p_tyNtParamCurr.tyProdRcpWidth.diMax THEN
			bChkMagLmtOk	:= FALSE;
			bChkMagLmtNG	:= TRUE;
			sAddMsg		:= 'Maximum Board Width Upper Limit ';
		ELSE

			bChkMagLmtOk	:= TRUE;
			bChkMagLmtNG	:= FALSE;
			sAddMsg		:= '';

		END_IF
	ELSE

		bChkMagLmtOk	:= FALSE;
		bChkMagLmtNG	:= FALSE;
	END_IF

	//Update LCS Enable
	tyTagNm.bMngRcpEn		:= p_bLinkNtParamLCSManageRcpPrep AND p_bLinkMcParamLCSManageRcpEn;
	tyTagNm.bLFEn			:= p_bLinkNtParamLCSLFPrep AND p_bLinkMcParamLCSLFEn;
	tyTagNm.bLiveData		:= p_bLinkNtParamLCSLiveDatPrep AND p_bLinkMcParamLCSLiveDatEn;

	//tyTagNm.usiBrdStatus = 0 (Machine Empty)
	//tyTagNm.usiBrdStatus = 1 (Machine Not Empty)
	IF p_eLinkNtParamProjMag = ULMagDual THEN
		tyTagNm.usiBrdStatus	:= BOOL_TO_USINT(NOT(p_bLinkPshrConvHvBrd = FALSE AND p_bLinkBffr1MagRemoved = TRUE AND p_bLinkBffr2MagRemoved = TRUE));
	ELSIF p_eLinkNtParamProjMag = ULMagTriple THEN
		tyTagNm.usiBrdStatus	:= BOOL_TO_USINT(NOT(p_bLinkPshrConvHvBrd = FALSE AND p_bLinkBffr1MagRemoved = TRUE AND p_bLinkBffr2MagRemoved = TRUE AND p_bLinkBffr3MagRemoved = TRUE));
	END_IF

	//Action
	IF tyTagNm.eAct = LCSActRunProd THEN

		bLFRun		:= TRUE;
		bMngRcpRun	:= FALSE;

	ELSIF (tyTagNm.eAct = LCSActAddProd)
		OR (tyTagNm.eAct = LCSActAddMultiProd)
		OR (tyTagNm.eAct = LCSActEditProd)
		OR (tyTagNm.eAct = LCSActEditMultiProd)
		OR (tyTagNm.eAct = LCSActOverWriteProd)
		OR (tyTagNm.eAct = LCSActOverWriteMultiProd)
		OR (tyTagNm.eAct = LCSActDelProd)
		OR (tyTagNm.eAct = LCSActDelMultiProd)
		OR (tyTagNm.eAct = LCSActUploadProd)
		OR (tyTagNm.eAct = LCSActUploadMultiProd)
		OR (tyTagNm.eAct = LCSActOverWriteMag)
		OR (tyTagNm.eAct = LCSActDelMag)
		OR (tyTagNm.eAct = LCSActUploadMag)
		THEN

		bLFRun		:= FALSE;
		bMngRcpRun	:= TRUE;

	ELSIF tyTagNm.eAct = LCSActIdle THEN

		bLFRun		:= FALSE;
		bMngRcpRun	:= FALSE;

	END_IF

	IF bLFRun = TRUE THEN
		eLCSLF_LCSAct			:= tyTagNm.eAct;
		tyLCSLF_LCSProdRcpInfo	:= tyTagNm.tyProdRcpInfo;

		tyLCSLF_LCSProdRcpInfo.bTopToBtm	:= INT_TO_BOOL(tyTagNm.iTopToBtm);

		sLastModifiedTemp	:= CONCAT('DT#' , tyTagNm.sLastModified);
		tyLCSLF_LCSProdRcpInfo.dtLastModified	:= STRING_TO_DT(sLastModifiedTemp);

		tyTagNm.eStat		:= p_eLCSLF_PLCStat;
		tyTagNm.udiStatus	:= p_udiLCSLF_PLCStatus;

		IF tyTagNm.udiStatus > 0 AND tyTagNm.udiStatus < 65534 THEN
			tyTagNm.sErrMsg	:= a_tyAlmText[tyTagNm.udiStatus].sAlmText;

			IF tyTagNm.udiStatus = 10010 OR tyTagNm.udiStatus = 10011 THEN
				tyTagNm.sErrMsg	:= CONCAT(sAddMsg , tyTagNm.sErrMsg);
			END_IF
		END_IF

	ELSIF bMngRcpRun = TRUE THEN
		eLCSMngRcp_LCSAct	:= tyTagNm.eAct;
		IF tyTagNm.tyProdRcpInfo.diBrdPerSlt <1 THEN
			tyTagNm.tyProdRcpInfo.diBrdPerSlt := 1;
		END_IF
		tyTagNm.eStat		:= p_eLCSMngRcp_PLCStat;
		tyTagNm.udiStatus	:= p_udiLCSMngRcp_PLCStatus;

		IF tyTagNm.udiStatus > 0 AND tyTagNm.udiStatus < 65534 THEN
			tyTagNm.sErrMsg	:= a_tyAlmText[tyTagNm.udiStatus].sAlmText;

			IF tyTagNm.udiStatus = 10010 OR tyTagNm.udiStatus = 10011 THEN
				tyTagNm.sErrMsg	:= CONCAT(sAddMsg , tyTagNm.sErrMsg);
			END_IF
		END_IF

		IF tyTagNm.eAct = LCSActUploadProd THEN
			IF tyTagNm.udiStatus = 0 THEN
				tyTagNm.tyProdRcpInfo	:= p_tyLCSMngRcp_PLCProdRcpInfo;

				tyTagNm.iTopToBtm	:= BOOL_TO_INT(tyLCSMngRcp_LCSProdRcpInfo.bTopToBtm);

				tyTagNm.sLastModified	:= DT_TO_STRING(tyLCSMngRcp_LCSProdRcpInfo.dtLastModified);
				tyTagNm.sLastModified	:= RIGHT(tyTagNm.sLastModified , (LEN(tyTagNm.sLastModified) - 3));

			ELSE
				tyLCSMngRcp_LCSProdRcpInfo	:= tyTagNm.tyProdRcpInfo;

				tyLCSMngRcp_LCSProdRcpInfo.bTopToBtm	:= INT_TO_BOOL(tyTagNm.iTopToBtm);
				tyLCSMngRcp_LCSProdRcpInfo.diWidthInUM2 := tyTagNm.tyProdRcpInfo.diWidthInUM;

				sLastModifiedTemp	:= CONCAT('DT#' , tyTagNm.sLastModified);
				tyLCSMngRcp_LCSProdRcpInfo.dtLastModified	:= STRING_TO_DT(sLastModifiedTemp);

			END_IF

		ELSIF tyTagNm.eAct = LCSActUploadMultiProd THEN
			iLCSMngRcp_LCSIdxStat	:= tyTagNm.iIdxAct;

			tyTagNm.iIdxStat		:= p_iLCSMngRcp_PLCIdxAct;

			tyTagNm.tyProdRcpInfo	:= p_tyLCSMngRcp_PLCProdRcpInfo;

			tyTagNm.iTopToBtm	:= BOOL_TO_INT(tyLCSMngRcp_LCSProdRcpInfo.bTopToBtm);

			tyTagNm.sLastModified	:= DT_TO_STRING(tyLCSMngRcp_LCSProdRcpInfo.dtLastModified);
			tyTagNm.sLastModified	:= RIGHT(tyTagNm.sLastModified , (LEN(tyTagNm.sLastModified) - 3));
		ELSIF tyTagNm.eAct = LCSActUploadMag THEN
			IF tyTagNm.udiStatus = 0 THEN
				tyTagNm.tyMagRcpInfo	:= p_tyLCSMngRcp_PLCMagRcpInfo;

				tyTagNm.iTopToBtm	:= BOOL_TO_INT(tyLCSMngRcp_LCSProdRcpInfo.bTopToBtm);

				tyTagNm.sLastModified	:= DT_TO_STRING(tyLCSMngRcp_LCSProdRcpInfo.dtLastModified);
				tyTagNm.sLastModified	:= RIGHT(tyTagNm.sLastModified , (LEN(tyTagNm.sLastModified) - 3));

			ELSE
				tyLCSMngRcp_LCSMagRcpInfo	:= tyTagNm.tyMagRcpInfo;

				sLastModifiedTemp	:= CONCAT('DT#' , tyTagNm.sLastModified);
				tyLCSMngRcp_LCSMagRcpInfo.dtLastModified	:= STRING_TO_DT(sLastModifiedTemp);

			END_IF
		ELSE
			iLCSMngRcp_LCSIdxAct		:= tyTagNm.iIdxAct;
			tyLCSMngRcp_LCSProdRcpInfo	:= tyTagNm.tyProdRcpInfo;
			tyLCSMngRcp_LCSMagRcpInfo   := tyTagNm.tyMagRcpInfo;

			tyLCSMngRcp_LCSProdRcpInfo.bTopToBtm	:= INT_TO_BOOL(tyTagNm.iTopToBtm);
			tyLCSMngRcp_LCSProdRcpInfo.diWidthInUM2 := tyTagNm.tyProdRcpInfo.diWidthInUM;

			sLastModifiedTemp	:= CONCAT('DT#' , tyTagNm.sLastModified);
			tyLCSMngRcp_LCSProdRcpInfo.dtLastModified	:= STRING_TO_DT(sLastModifiedTemp);

			tyTagNm.iIdxStat	:= p_iLCSMngRcp_PLCIdxStat;

		END_IF

	ELSE

		eLCSLF_LCSAct		:= LCSActIdle;
		eLCSMngRcp_LCSAct	:= LCSActIdle;
		tyTagNm.eStat		:= LCSActIdle;
		tyTagNm.udiStatus	:= 65534;
		tyTagNm.sErrMsg		:= '';

	END_IF

END_ACTION
```

#### Act_Background_LiveData.st - Do Not Change!!!
```iecst
(** 2019-07-10 **)
ACTION Act_Background_LiveData:

	IF p_bLinkNtParamLCSLiveDatPrep AND p_bLinkMcParamLCSLiveDatEn THEN

		tyTagNm.sCurrRcpNm	:= p_tyProdRcpCurrRcp.sRcpNm;
		tyTagNm.rCurrWidth	:= DINT_TO_REAL(p_tyProdRcpCurrRcp.diWidthInUM) / 1000;
		tyTagNm.usiMode		:= BOOL_TO_USINT(p_bLinkNtParamLCSLFPrep AND p_bLinkMcParamLCSLFEn);
		tyTagNm.sCurrMagRcpNm := p_tyMagRcpCurrRcp.sRcpNm; //LCS Added
		tyTagNm.tyCurrMagRcpParam := p_tyMagRcpCurrRcp; //LCS Added

		IF p_bError = TRUE THEN
			tyTagNm.eCurrOpsStatus	:= LCSOpsStatusError;
		ELSIF p_bWarning = TRUE OR p_bInfo = TRUE THEN
			tyTagNm.eCurrOpsStatus	:= LCSOpsStatusWarning;
		ELSIF p_bOpsRun = TRUE THEN
			tyTagNm.eCurrOpsStatus	:= LCSOpsStatusAuto;
		ELSIF p_bUIManual = TRUE THEN
			tyTagNm.eCurrOpsStatus	:= LCSOpsStatusManual;
		ELSE
			tyTagNm.eCurrOpsStatus	:= LCSOpsStatusStop;
		END_IF

	END_IF

END_ACTION
```

#### InputRef.var - Do Not Change!!!
```iecst
(*2019-06-12*)
(**)
(*General*)
VAR
	p_bPrep : REFERENCE TO BOOL;
	p_bEn : REFERENCE TO BOOL;
	p_bDis : REFERENCE TO BOOL;
END_VAR
(**)
(*Configuration*)
VAR
	p_eLCSMngRcp_PLCStat : REFERENCE TO eLCSAction;
	p_udiLCSMngRcp_PLCStatus : REFERENCE TO UDINT;
	p_iLCSMngRcp_PLCIdxAct : REFERENCE TO INT;
	p_iLCSMngRcp_PLCIdxStat : REFERENCE TO INT;
	p_tyLCSMngRcp_PLCProdRcpInfo : REFERENCE TO tyProdRcpParam;
	p_eLCSLF_PLCStat : REFERENCE TO eLCSAction;
	p_udiLCSLF_PLCStatus : REFERENCE TO UDINT;
	p_bLCSMngRcpChkLmt : REFERENCE TO BOOL;
	p_bLCSLFChkLmt : REFERENCE TO BOOL;
	p_bOpsRun : REFERENCE TO BOOL;
	p_bError : REFERENCE TO BOOL;
	p_bWarning : REFERENCE TO BOOL;
	p_bInfo : REFERENCE TO BOOL;
	p_bUIManual : REFERENCE TO BOOL;
	p_tyProdRcpCurrRcp : REFERENCE TO tyProdRcpParam;
	p_tyNtParamCurr : REFERENCE TO tyNtParam;
	p_sProgNm : REFERENCE TO STRING[15];
	p_bNtSettingsLoadDone : REFERENCE TO BOOL;
	p_tyMagRcpCurrRcp : REFERENCE TO tyMagRcpParam;
	p_tyLCSMngRcp_PLCMagRcpInfo : REFERENCE TO tyMagRcpParam;
	p_bLCSMngMagRcpChkLmt : REFERENCE TO BOOL;
END_VAR
```

#### Local.var - Do Not Change!!!
```iecst
(*2019-06-12*)
(**)
(*Local Action, State & Status*)
(**)
(*Local Alarm*)
VAR
	a_tyAlmText : ARRAY[10000..10099] OF tyAlmTxt := [(sAlmText:='LCS Disable'),(sAlmText:='LCS Manage Recipe Disabled'),(sAlmText:='LCS Leader Follower Disabled'),7(0),(sAlmText:='Out Of Range While Accepting New Recipe'),(sAlmText:='Out Of Range While Managing Product'),(sAlmText:='Recipe Name Empty While Adding Product'),(sAlmText:='Recipe List Full While Adding Product'),(sAlmText:='Recipe Name Exist While Adding Product'),(sAlmText:='Recipe Program Error While Adding Product'),(sAlmText:='Check Limit Error While Adding Multiple Product'),(sAlmText:='Recipe Name Empty While Adding Multiple Product'),(sAlmText:='Recipe List Full While Adding Multiple Product'),(sAlmText:='Recipe Name Exist While Adding Multiple Product'),(sAlmText:='Recipe Program Error While Adding Multiple Product'),(sAlmText:='Check Limit Error While Editing Product'),(sAlmText:='Recipe Name Empty While Editing Product'),(sAlmText:='Recipe Name Not Exist While Editing Product'),(sAlmText:='Recipe Program Error While Editing Product'),(sAlmText:='Check Limit Error While Editing Multiple Product'),(sAlmText:='Recipe Name Empty While Editing Multiple Product'),(sAlmText:='Recipe Name Not Exist While Editing Multiple Product'),(sAlmText:='Recipe Program Error While Editing Multiple Product'),(sAlmText:='Check Limit Error While Overwriting Product'),(sAlmText:='Recipe Name Empty While Overwriting Product'),(sAlmText:='Recipe List Full While Overwriting Product'),(sAlmText:='Recipe Program Error While Overwriting Product'),(sAlmText:='Check Limit Error While Overwriting Multiple Product'),(sAlmText:='Recipe Name Empty While Overwriting Multiple Product'),(sAlmText:='Recipe List Full While Overwriting Multiple Product'),(sAlmText:='Recipe Program Error While Overwriting Multiple Product'),(sAlmText:='Check Limit Error While Deleting Product'),(sAlmText:='Recipe Name Empty While Deleting Product'),(sAlmText:='Recipe Name Not Exist While Deleting Product'),(sAlmText:='Recipe Program Error While Deleting Product'),(sAlmText:='Check Limit Error While Deleting Multiple Product'),(sAlmText:='Recipe Name Empty While Deleting Multiple Product'),(sAlmText:='Recipe Name Not Exist While Deleting Multiple Product'),(sAlmText:='Recipe Program Error While Deleting Multiple Product'),(sAlmText:='Recipe Name Empty While Uploading Product'),(sAlmText:='Recipe Name Not Exist While Uploading Product'),(sAlmText:='Recipe Program Error While Uploading Product'),(sAlmText:='Get Recipe Info Error While Editing Product'),(sAlmText:='Local Recipe Is Latest Compare With LCS Recipe While Editing Product'),(sAlmText:='Local Recipe Is Latest Compare With LCS Recipe While Editing Multiple Product'),(sAlmText:='Get Recipe Info Error While Editing Multiple Product'),48(0)];
END_VAR
(**)
(*Local Output*)
VAR
	eLCSMngRcp_LCSAct : eLCSAction;
	iLCSMngRcp_LCSIdxAct : INT;
	iLCSMngRcp_LCSIdxStat : INT;
	tyLCSMngRcp_LCSProdRcpInfo : tyProdRcpParam;
	eLCSLF_LCSAct : eLCSAction;
	tyLCSLF_LCSProdRcpInfo : tyProdRcpParam;
	bChkLmtOK : BOOL;
	bChkLmtNG : BOOL;
	bChkMagLmtOk : BOOL;
	bChkMagLmtNG : BOOL;
END_VAR
(**)
(*Local Input*)
VAR
	bPrep : BOOL := TRUE;
	bEn : BOOL := TRUE;
	bDis : BOOL := FALSE;
	eLCSMngRcp_PLCStat : eLCSAction;
	udiLCSMngRcp_PLCStatus : UDINT;
	iLCSMngRcp_PLCIdxAct : INT;
	iLCSMngRcp_PLCIdxStat : INT;
	tyLCSMngRcp_PLCProdRcpInfo : tyProdRcpParam;
	eLCSLF_PLCStat : eLCSAction;
	udiLCSLF_PLCStatus : UDINT;
	bLCSMngRcpChkLmt : BOOL;
	bLCSLFChkLmt : BOOL;
	bOpsRun : BOOL;
	bError : BOOL;
	bWarning : BOOL;
	bInfo : BOOL;
	bUIManual : BOOL;
	tyProdRcpCurrRcp : tyProdRcpParam;
	tyNtParamCurr : tyNtParam;
	sProgNm : STRING[15] := 'LCS';
	bNtSettingsLoadDone : BOOL := TRUE;
END_VAR
(**)
(*Local*)
VAR
	udi : UDINT;
	udiFlagNo : UDINT;
	bInitDone : BOOL;
	bInitialDone : BOOL;
	tyTagNm : tyLCSTagNm;
	bLFRun : BOOL;
	bMngRcpRun : BOOL;
	sLastModifiedTemp : STRING[80];
	sAddMsg : STRING[80];
	udiModuleNum : UDINT := 4001;
	tyLCSMngRcp_LCSMagRcpInfo : tyMagRcpParam;
END_VAR
```

### LCSMngRcp.var - Change By Project
```iecst
(*2019-04-24*)
(**)
(*Action & State & Status*)
VAR
	p_LCSMngRcpStat : UDINT;
	p_LCSMngRcpStatus : UDINT;
	p_LCSMngRcpStatTxt : UDINT;
END_VAR
(**)
(*Alarm*)
VAR
	p_LCSMngRcpAlmData : UDINT;
END_VAR
(**)
(*Output*)
VAR
	p_LCSMngRcp_PLCStatus : UDINT;
	p_LCSMngRcp_PLCIdxAct : UDINT;
	p_LCSMngRcp_PLCIdxStat : UDINT;
	p_LCSMngRcp_PLCProdRcpInfo : UDINT;
	p_LCSMngRcpProdRcpAct : UDINT;
	p_LCSMngRcpProdRcpInfoIn : UDINT;
	p_LCSMngRcpChkLmt : UDINT;
	p_LCSMngRcpMagRcpAct : UDINT;
	p_LCSMngRcpMagRcpInfoIn : UDINT;
	p_LCSMngRcp_PLCMagRcpInfo : UDINT;
	p_LCSMngMagRcpChkLmt : UDINT;
END_VAR
```

### Program Logical/LCS/LCSMngRcp (IEC) - 1.00.0 - NtRecipe v5.00.0 , NtFileIO v5.00.0

#### InputRef.var
```iecst
(*2019-04-24*)
(**)
(*General*)
VAR
	p_eAct : REFERENCE TO eLCSAction;
	p_udiRstErr : REFERENCE TO UDINT;
	p_bPrep : REFERENCE TO BOOL;
	p_bEn : REFERENCE TO BOOL;
	p_bDis : REFERENCE TO BOOL;
END_VAR
(**)
(*Configuration*)
VAR
	p_bProdRcpNmExist : REFERENCE TO BOOL;
	p_bProdRcpNmNotExist : REFERENCE TO BOOL;
	p_bProdRcpNmEmpty : REFERENCE TO BOOL;
	p_bProdRcpListFull : REFERENCE TO BOOL;
	pa_tyProdRcpCurrList : REFERENCE TO ARRAY[1..c_udiProdRcpMax] OF tyProdRcpParam;
	p_tyProdRcpInfoOut : REFERENCE TO tyProdRcpParam;
	p_tyProdRcpCurrRcp : REFERENCE TO tyProdRcpParam;
	p_eProdRcpStat : REFERENCE TO eProdRcpAction;
	p_eProdRcpStatus : REFERENCE TO eFBStatus;
	p_sMcParamProdSelRcpNm : REFERENCE TO STRING[15];
	p_diMcParamProdSelWidth : REFERENCE TO DINT;
	p_iLCSIdxAct : REFERENCE TO INT;
	p_iLCSIdxStat : REFERENCE TO INT;
	p_tyLCSProdRcpInfo : REFERENCE TO tyProdRcpParam;
	p_bChkLmtOK : REFERENCE TO BOOL;
	p_bChkLmtNG : REFERENCE TO BOOL;
	p_sProgNm : REFERENCE TO STRING[15];
	p_bNtSettingsLoadDone : REFERENCE TO BOOL;
	p_tyLCSMagRcpInfo : REFERENCE TO tyMagRcpParam;
	p_eMagRcpStat : REFERENCE TO eMagRcpAction;
	p_eMagRcpStatus : REFERENCE TO eFBStatus;
	p_bMagRcpNmEmpty : REFERENCE TO BOOL;
	p_bMagRcpNmNotExist : REFERENCE TO BOOL;
	p_tyMagRcpInfoOut : REFERENCE TO tyMagRcpParam;
	p_bChkMagLmtOK : REFERENCE TO BOOL;
	p_bChkMagLmtNG : REFERENCE TO BOOL;
	p_bMagRcpListFull : REFERENCE TO BOOL;
END_VAR
```

#### Local.var
```iecst
(*2019-04-30*)
(**)
(*Local Action, State & Status*)
VAR
	eAct : eLCSAction := LCSActIdle;
	eStat : eLCSAction := LCSActIdle;
	eStatus : eFBStatus := Idle;
	udiStatus : UDINT := 0;
	sStatTxt : STRING[200] := '';
	a_sStatText : ARRAY[0..50] OF STRING[200] := ['Idling','Adding Product','Adding Multiple Products','Editing Product','Editing Multiple Products','OverWrite Product','OverWrite Multiple Products','Deleting Product','Deleting Multiple Products','Running LCS Product','Uploading Product','Uploading Multiple Products',39('')];
END_VAR
(**)
(*Local Alarm*)
VAR
	tyAlmData : tyAlmDat;
	a_tyAlmText : ARRAY[10000..10099] OF tyAlmTxt;
END_VAR
(**)
(*Local Output*)
VAR
	udiPLCStatus : UDINT;
	iPLCIdxAct : INT;
	iPLCIdxStat : INT;
	tyPLCProdRcpInfo : tyProdRcpParam;
	eProdRcpAct : eProdRcpAction;
	tyProdRcpInfoIn : tyProdRcpParam;
	tyPLCMagRcpInfo : tyMagRcpParam;
	eMagRcpAct : eMagRcpAction;
	tyMagRcpInfoIn : tyMagRcpParam;
	bChkLmt : BOOL;
	bChkMagLmt : BOOL;
END_VAR
(**)
(*Local Input*)
VAR
	udiRstErr : UDINT := 0;
	bPrep : BOOL := TRUE;
	bEn : BOOL := TRUE;
	bDis : BOOL := FALSE;
	bProdRcpNmExist : BOOL;
	bProdRcpNmNotExist : BOOL;
	bProdRcpNmEmpty : BOOL;
	bProdRcpListFull : BOOL;
	a_tyProdRcpCurrList : ARRAY[1..c_udiProdRcpMax] OF tyProdRcpParam;
	tyProdRcpInfoOut : tyProdRcpParam;
	tyProdRcpCurrRcp : tyProdRcpParam;
	eProdRcpStat : eProdRcpAction;
	eProdRcpStatus : eFBStatus;
	sMcParamProdSelRcpNm : STRING[15];
	diMcParamProdSelWidth : DINT;
	iLCSIdxAct : INT;
	iLCSIdxStat : INT;
	tyLCSProdRcpInfo : tyProdRcpParam;
	bChkLmtOK : BOOL;
	bChkLmtNG : BOOL;
	sProgNm : STRING[15] := 'LCSMngRcp';
	bNtSettingsLoadDone : BOOL := TRUE;
END_VAR
(**)
(*Local*)
VAR
	bRstErr : BOOL;
	udiRstErrOld : UDINT;
	bInitDone : BOOL;
	bInitialDone : BOOL;
	usiStep : USINT;
	udiModuleNum : UDINT := 4201;
END_VAR
```

#### Act_InitGlobal.st
```iecst
(** 2019-04-24 **)
ACTION Act_InitGlobal:

	(* Always Change If Project Change *)

	//Pass Data To Link
	p_bLinkStartupRun ACCESS p_StartupRun;

	//Pass Data To Internal Use
	p_eAct ACCESS p_LCS_LCSMngRcp_LCSAct;
	p_udiRstErr ACCESS p_RstErrReset;
	p_bPrep ACCESS p_NtParamLCSManageRcpPrep;
	p_bEn ACCESS p_McParamLCSManageRcpEn;
	p_bProdRcpNmExist ACCESS p_ProdRcpNmExist;
	p_bProdRcpNmNotExist ACCESS p_ProdRcpNmNotExist;
	p_bProdRcpNmEmpty ACCESS p_ProdRcpNmEmpty;
	p_bProdRcpListFull ACCESS p_ProdRcpListFull;
	pa_tyProdRcpCurrList ACCESS p_ProdRcpCurrList;
	p_tyProdRcpInfoOut ACCESS p_ProdRcpInfoOut;
	p_tyProdRcpCurrRcp ACCESS p_ProdRcpCurrRcp0;
	p_eProdRcpStat ACCESS p_ProdRcpStat;
	p_eProdRcpStatus ACCESS p_ProdRcpStatus;
	p_sMcParamProdSelRcpNm ACCESS p_ProdRcpCurrRcp0Nm;
	p_diMcParamProdSelWidth ACCESS p_ProdRcpCurrRcp0Width;
	p_iLCSIdxAct ACCESS p_LCS_LCSMngRcp_LCSIdxAct;
	p_iLCSIdxStat ACCESS p_LCS_LCSMngRcp_LCSIdxStat;
	p_tyLCSProdRcpInfo ACCESS p_LCS_LCSMngRcp_LCSProdRcpInfo;
	p_bChkLmtOK ACCESS p_LCSChkLmtOK;
	p_bChkLmtNG ACCESS p_LCSChkLmtNG;
	p_sProgNm ACCESS p_NtParamLCSMngRcpProgNm;
	p_bNtSettingsLoadDone ACCESS p_StartupNtSettingsLoadDone;

	p_tyLCSMagRcpInfo ACCESS p_LCS_LCSMngRcp_LCSMagRcpInfo;
	p_eMagRcpStat ACCESS p_MagRcpStat;
	p_eMagRcpStatus ACCESS p_MagRcpStatus;
	p_bMagRcpNmEmpty ACCESS p_MagRcpNmEmpty;
	p_bMagRcpNmNotExist ACCESS p_MagRcpNmNotExist;
	p_bMagRcpListFull ACCESS p_MagRcpListFull;
	p_tyMagRcpInfoOut ACCESS p_MagRcpInfoOut;
	p_bChkMagLmtOK ACCESS p_LCSChkMagLmtOK;
	p_bChkMagLmtNG ACCESS p_LCSChkMagLmtNG;
	(* Always Change If Project Change *)

END_ACTION
```

#### Act_Main.st
```iecst
(** 2019-04-24 **)
ACTION Act_Main:

	//Main
	CASE eStat OF

		LCSActIdle:
			IF eStatus <> Idle THEN	//Reset Data
				//Private
				eProdRcpAct		:= ProdRcpActIdle;
				usiStep			:= 0;
				iPLCIdxAct		:= 0;
				iPLCIdxStat		:= 0;
				bChkLmt			:= FALSE;

				sStatTxt		:= a_sStatText[eStat];

			END_IF

			eStatus			:= Idle;
			udiPLCStatus	:= 65534;

		LCSActAddProd:
			IF eStatus = Idle OR eStatus = Busy THEN

				eStatus			:= Busy;
				udiPLCStatus	:= 65535;

				sStatTxt	:= a_sStatText[eStat];

				CASE usiStep OF
					0:
						bChkLmt	:= TRUE;

						IF p_bChkLmtOK = TRUE THEN
							usiStep			:= 1;
						ELSIF p_bChkLmtNG = TRUE THEN
							eStatus			:= Done;
							udiPLCStatus	:= 10011;	//Out Of Range While Managing Product
						END_IF

					1:
						tyProdRcpInfoIn	:= p_tyLCSProdRcpInfo;
						eProdRcpAct		:= ProdRcpActAdd;

						IF (p_eProdRcpStat = ProdRcpActAdd) AND (p_eProdRcpStatus = Done) THEN
							eStatus		:= Done;

							IF p_bProdRcpNmEmpty = TRUE THEN
								udiPLCStatus	:= 10012;	//Recipe Name Empty While Adding Product
							ELSIF p_bProdRcpListFull = TRUE THEN
								udiPLCStatus	:= 10013;	//Recipe List Full While Adding Product
							ELSIF p_bProdRcpNmExist = TRUE THEN
								udiPLCStatus	:= 10014;	//Recipe Name Exist While Adding Product
							ELSE
								udiPLCStatus	:= 0;
							END_IF

							eProdRcpAct	:= ProdRcpActIdle;

						ELSIF p_eProdRcpStatus = Error THEN
							eStatus			:= Done;
							udiPLCStatus	:= 10015;	//Recipe Program Error While Adding Product
						END_IF

				END_CASE

			END_IF

		LCSActAddMultiProd:
			IF eStatus = Idle OR eStatus = Busy THEN

				eStatus			:= Busy;
				udiPLCStatus	:= 65535;

				sStatTxt	:= a_sStatText[eStat];

				IF (p_iLCSIdxAct <> 0) THEN
					IF p_iLCSIdxAct <> iPLCIdxStat THEN

						CASE usiStep OF
							0:
								bChkLmt	:= TRUE;

								IF p_bChkLmtOK = TRUE THEN
									usiStep			:= 1;
								ELSIF p_bChkLmtNG = TRUE THEN
									eStatus			:= Done;
									udiPLCStatus	:= 10016;	//Check Limit Error While Adding Multiple Product
								END_IF

							1:
								tyProdRcpInfoIn	:= p_tyLCSProdRcpInfo;
								eProdRcpAct		:= ProdRcpActAdd;

								IF (p_eProdRcpStat = ProdRcpActAdd) AND (p_eProdRcpStatus = Done) THEN
									IF p_bProdRcpNmEmpty = TRUE THEN
										eStatus			:= Done;
										udiPLCStatus	:= 10017;	//Recipe Name Empty While Adding Multiple Product
									ELSIF p_bProdRcpListFull = TRUE THEN
										eStatus			:= Done;
										udiPLCStatus	:= 10018;	//Recipe List Full While Adding Multiple Product
									ELSIF p_bProdRcpNmExist = TRUE THEN
										eStatus			:= Done;
										udiPLCStatus	:= 10019;	//Recipe Name Exist While Adding Multiple Product
									ELSE
										iPLCIdxStat	:= p_iLCSIdxAct;
										usiStep		:= 0;
									END_IF

									eProdRcpAct	:= ProdRcpActIdle;

								ELSIF p_eProdRcpStatus = Error THEN
									eStatus			:= Done;
									udiPLCStatus	:= 10020;	//Recipe Program Error While Adding Multiple Product
								END_IF

						END_CASE

					END_IF

				ELSE
					eStatus			:= Done;
					udiPLCStatus	:= 0;

				END_IF

			END_IF

		LCSActEditProd:
			IF eStatus = Idle OR eStatus = Busy THEN

				eStatus			:= Busy;
				udiPLCStatus	:= 65535;

				sStatTxt	:= a_sStatText[eStat];

				CASE usiStep OF
					0:
						bChkLmt	:= TRUE;

						IF p_bChkLmtOK = TRUE THEN
							usiStep			:= 1;
						ELSIF p_bChkLmtNG = TRUE THEN
							eStatus			:= Done;
							udiPLCStatus	:= 10021;	//Check Limit Error While Editing Product
						END_IF

					1:
						eProdRcpAct	:= ProdRcpActGetInfo;

						IF (p_eProdRcpStat = ProdRcpActGetInfo) AND (p_eProdRcpStatus = Done) THEN

							IF p_tyProdRcpInfoOut.dtLastModified > p_tyLCSProdRcpInfo.dtLastModified THEN
								eStatus			:= Done;
								udiPLCStatus	:= 10049;	//Local Recipe Is Latest Compare With LCS Recipe While Editing Product
							ELSE
								eProdRcpAct	:= ProdRcpActIdle;
								usiStep		:= 2;
							END_IF

						ELSIF p_eProdRcpStatus = Error THEN
							eStatus			:= Done;
							udiPLCStatus	:= 10048;	//Get Recipe Info Error While Editing Product
						END_IF

					2:
						tyProdRcpInfoIn	:= p_tyLCSProdRcpInfo;
						eProdRcpAct		:= ProdRcpActEdit;

						IF (p_eProdRcpStat = ProdRcpActEdit) AND (p_eProdRcpStatus = Done) THEN
							eStatus		:= Done;

							IF p_bProdRcpNmEmpty = TRUE THEN
								udiPLCStatus	:= 10022;	//Recipe Name Empty While Editing Product
							ELSIF p_bProdRcpNmNotExist = TRUE THEN
								udiPLCStatus	:= 10023;	//Recipe Name Not Exist While Editing Product
							ELSE
								udiPLCStatus	:= 0;
							END_IF

							eProdRcpAct	:= ProdRcpActIdle;

						ELSIF p_eProdRcpStatus = Error THEN
							eStatus			:= Done;
							udiPLCStatus	:= 10024;	//Recipe Program Error While Editing Product
						END_IF

				END_CASE

			END_IF

		LCSActEditMultiProd:
			IF eStatus = Idle OR eStatus = Busy THEN

				eStatus			:= Busy;
				udiPLCStatus	:= 65535;

				sStatTxt	:= a_sStatText[eStat];

				IF (p_iLCSIdxAct <> 0) THEN
					IF p_iLCSIdxAct <> iPLCIdxStat THEN

						CASE usiStep OF
							0:
								bChkLmt	:= TRUE;

								IF p_bChkLmtOK = TRUE THEN
									usiStep			:= 1;
								ELSIF p_bChkLmtNG = TRUE THEN
									eStatus			:= Done;
									udiPLCStatus	:= 10025;	//Check Limit Error While Editing Multiple Product
								END_IF

							1:
								eProdRcpAct	:= ProdRcpActGetInfo;

								IF (p_eProdRcpStat = ProdRcpActGetInfo) AND (p_eProdRcpStatus = Done) THEN

									IF p_tyProdRcpInfoOut.dtLastModified > p_tyLCSProdRcpInfo.dtLastModified THEN
										eStatus			:= Done;
										udiPLCStatus	:= 10050;	//Local Recipe Is Latest Compare With LCS Recipe While Editing Multiple Product
									ELSE
										eProdRcpAct	:= ProdRcpActIdle;
										usiStep		:= 2;
									END_IF

								ELSIF p_eProdRcpStatus = Error THEN
									eStatus			:= Done;
									udiPLCStatus	:= 10051;	//Get Recipe Info Error While Editing Multiple Product
								END_IF

							2:
								tyProdRcpInfoIn	:= p_tyLCSProdRcpInfo;
								eProdRcpAct		:= ProdRcpActEdit;

								IF (p_eProdRcpStat = ProdRcpActEdit) AND (p_eProdRcpStatus = Done) THEN
									IF p_bProdRcpNmEmpty = TRUE THEN
										eStatus			:= Done;
										udiPLCStatus	:= 10026;	//Recipe Name Empty While Editing Multiple Product
									ELSIF p_bProdRcpNmNotExist = TRUE THEN
										eStatus			:= Done;
										udiPLCStatus	:= 10027;	//Recipe Name Not Exist While Editing Multiple Product
									ELSE
										iPLCIdxStat	:= p_iLCSIdxAct;
										usiStep		:= 0;
									END_IF

									eProdRcpAct	:= ProdRcpActIdle;

								ELSIF p_eProdRcpStatus = Error THEN
									eStatus			:= Done;
									udiPLCStatus	:= 10028;	//Recipe Program Error While Editing Multiple Product
								END_IF

						END_CASE

					END_IF

				ELSE
					eStatus			:= Done;
					udiPLCStatus	:= 0;

				END_IF

			END_IF

		LCSActOverWriteProd:
			IF eStatus = Idle OR eStatus = Busy THEN

				eStatus			:= Busy;
				udiPLCStatus	:= 65535;

				sStatTxt	:= a_sStatText[eStat];

				CASE usiStep OF
					0:
						bChkLmt	:= TRUE;

						IF p_bChkLmtOK = TRUE THEN
							usiStep			:= 1;
						ELSIF p_bChkLmtNG = TRUE THEN
							eStatus			:= Done;
							udiPLCStatus	:= 10029;	//Check Limit Error While Overwriting Product
						END_IF

					1:
						tyProdRcpInfoIn	:= p_tyLCSProdRcpInfo;
						eProdRcpAct		:= ProdRcpActAddEdit;

						IF (p_eProdRcpStat = ProdRcpActAddEdit) AND (p_eProdRcpStatus = Done) THEN
							eStatus		:= Done;

							IF p_bProdRcpNmEmpty = TRUE THEN
								udiPLCStatus	:= 10030;	//Recipe Name Empty While Overwriting Product
							ELSIF p_bProdRcpListFull = TRUE THEN
								udiPLCStatus	:= 10031;	//Recipe List Full While Overwriting Product
							ELSE
								udiPLCStatus	:= 0;
							END_IF

							eProdRcpAct	:= ProdRcpActIdle;

						ELSIF p_eProdRcpStatus = Error THEN
							eStatus			:= Done;
							udiPLCStatus	:= 10032;	//Recipe Program Error While Overwriting Product
						END_IF

				END_CASE

			END_IF

		LCSActOverWriteMultiProd:
			IF eStatus = Idle OR eStatus = Busy THEN

				eStatus			:= Busy;
				udiPLCStatus	:= 65535;

				sStatTxt	:= a_sStatText[eStat];

				IF (p_iLCSIdxAct <> 0) THEN
					IF p_iLCSIdxAct <> iPLCIdxStat THEN

						CASE usiStep OF
							0:
								bChkLmt	:= TRUE;

								IF p_bChkLmtOK = TRUE THEN
									usiStep			:= 1;
								ELSIF p_bChkLmtNG = TRUE THEN
									eStatus			:= Done;
									udiPLCStatus	:= 10033;	//Check Limit Error While Overwriting Multiple Product
								END_IF

							1:
								tyProdRcpInfoIn	:= p_tyLCSProdRcpInfo;
								eProdRcpAct		:= ProdRcpActAddEdit;

								IF (p_eProdRcpStat = ProdRcpActAddEdit) AND (p_eProdRcpStatus = Done) THEN
									IF p_bProdRcpNmEmpty = TRUE THEN
										eStatus			:= Done;
										udiPLCStatus	:= 10034;	//Recipe Name Empty While Overwriting Multiple Product
									ELSIF p_bProdRcpListFull = TRUE THEN
										eStatus			:= Done;
										udiPLCStatus	:= 10035;	//Recipe List Full While Overwriting Multiple Product
									ELSE
										iPLCIdxStat	:= p_iLCSIdxAct;
										usiStep		:= 0;
									END_IF

									eProdRcpAct	:= ProdRcpActIdle;

								ELSIF p_eProdRcpStatus = Error THEN
									eStatus			:= Done;
									udiPLCStatus	:= 10036;	//Recipe Program Error While Overwriting Multiple Product
								END_IF

						END_CASE

					END_IF

				ELSE
					eStatus			:= Done;
					udiPLCStatus	:= 0;

				END_IF

			END_IF

		LCSActDelProd:
			IF eStatus = Idle OR eStatus = Busy THEN

				eStatus			:= Busy;
				udiPLCStatus	:= 65535;

				sStatTxt	:= a_sStatText[eStat];

				CASE usiStep OF
					0:
						bChkLmt	:= TRUE;

						IF p_bChkLmtOK = TRUE THEN
							usiStep			:= 1;
						ELSIF p_bChkLmtNG = TRUE THEN
							eStatus			:= Done;
							udiPLCStatus	:= 10037;	//Check Limit Error While Deleting Product
						END_IF

					1:
						tyProdRcpInfoIn	:= p_tyLCSProdRcpInfo;
						eProdRcpAct		:= ProdRcpActDel;

						IF (p_eProdRcpStat = ProdRcpActDel) AND (p_eProdRcpStatus = Done) THEN
							eStatus		:= Done;

							IF p_bProdRcpNmEmpty = TRUE THEN
								udiPLCStatus	:= 10038;	//Recipe Name Empty While Deleting Product
							ELSIF p_bProdRcpNmNotExist = TRUE THEN
								udiPLCStatus	:= 10039;	//Recipe Name Not Exist While Deleting Product
							ELSE
								udiPLCStatus	:= 0;
							END_IF

							eProdRcpAct	:= ProdRcpActIdle;

						ELSIF p_eProdRcpStatus = Error THEN
							eStatus			:= Done;
							udiPLCStatus	:= 10040;	//Recipe Program Error While Deleting Product
						END_IF

				END_CASE

			END_IF

		LCSActDelMultiProd:
			IF eStatus = Idle OR eStatus = Busy THEN

				eStatus			:= Busy;
				udiPLCStatus	:= 65535;

				sStatTxt	:= a_sStatText[eStat];

				IF (p_iLCSIdxAct <> 0) THEN
					IF p_iLCSIdxAct <> iPLCIdxStat THEN

						CASE usiStep OF
							0:
								bChkLmt	:= TRUE;

								IF p_bChkLmtOK = TRUE THEN
									usiStep			:= 1;
								ELSIF p_bChkLmtNG = TRUE THEN
									eStatus			:= Done;
									udiPLCStatus	:= 10041;	//Check Limit Error While Deleting Multiple Product
								END_IF

							1:
								tyProdRcpInfoIn	:= p_tyLCSProdRcpInfo;
								eProdRcpAct		:= ProdRcpActDel;

								IF (p_eProdRcpStat = ProdRcpActDel) AND (p_eProdRcpStatus = Done) THEN
									IF p_bProdRcpNmEmpty = TRUE THEN
										eStatus			:= Done;
										udiPLCStatus	:= 10042;	//Recipe Name Empty While Deleting Multiple Product
									ELSIF p_bProdRcpNmNotExist = TRUE THEN
										eStatus			:= Done;
										udiPLCStatus	:= 10043;	//Recipe Name Not Exist While Deleting Multiple Product
									ELSE
										iPLCIdxStat	:= p_iLCSIdxAct;
										usiStep		:= 0;
									END_IF

									eProdRcpAct	:= ProdRcpActIdle;

								ELSIF p_eProdRcpStatus = Error THEN
									eStatus			:= Done;
									udiPLCStatus	:= 10044;	//Recipe Program Error While Deleting Multiple Product
								END_IF

						END_CASE

					END_IF

				ELSE
					eStatus			:= Done;
					udiPLCStatus	:= 0;

				END_IF

			END_IF

		LCSActUploadProd:
			IF eStatus = Idle OR eStatus = Busy THEN

				eStatus			:= Busy;
				udiPLCStatus	:= 65535;

				sStatTxt	:= a_sStatText[eStat];

				tyProdRcpInfoIn	:= p_tyLCSProdRcpInfo;
				eProdRcpAct		:= ProdRcpActGetInfo;

				IF (p_eProdRcpStat = ProdRcpActGetInfo) AND (p_eProdRcpStatus = Done) THEN
					eStatus		:= Done;

					IF p_bProdRcpNmEmpty = TRUE THEN
						udiPLCStatus	:= 10045;	//Recipe Name Empty While Uploading Product
					ELSIF p_bProdRcpNmNotExist = TRUE THEN
						eStatus			:= Done;
						udiPLCStatus	:= 10046;	//Recipe Name Not Exist While Uploading Product
					ELSE
						udiPLCStatus		:= 0;
						tyPLCProdRcpInfo	:= p_tyProdRcpInfoOut;
					END_IF

					eProdRcpAct	:= ProdRcpActIdle;

				ELSIF p_eProdRcpStatus = Error THEN
					eStatus			:= Done;
					udiPLCStatus	:= 10047;	//Recipe Program Error While Uploading Product
				END_IF

			END_IF

		LCSActUploadMultiProd:
			IF eStatus = Idle OR eStatus = Busy THEN

				eStatus			:= Busy;
				udiPLCStatus	:= 65535;

				sStatTxt	:= a_sStatText[eStat];

				IF (iPLCIdxAct = p_iLCSIdxStat) OR (iPLCIdxAct = 0) THEN

					IF pa_tyProdRcpCurrList[iPLCIdxAct + 1].sRcpNm <> '' THEN

						tyPLCProdRcpInfo	:= pa_tyProdRcpCurrList[iPLCIdxAct + 1];
						iPLCIdxAct			:= iPLCIdxAct + 1;

					ELSE

						eStatus			:= Done;
						udiPLCStatus	:= 0;
						iPLCIdxAct		:= 0;

					END_IF

				END_IF

			END_IF

		LCSActOverWriteMag:
			IF eStatus = Idle OR eStatus = Busy THEN

				eStatus			:= Busy;
				udiPLCStatus	:= 65535;

				sStatTxt	:= a_sStatText[eStat];

				CASE usiStep OF
					0:
						bChkMagLmt	:= TRUE;

						IF p_bChkMagLmtOK = TRUE THEN
							usiStep			:= 1;
						ELSIF p_bChkMagLmtNG = TRUE THEN
							eStatus			:= Done;
							udiPLCStatus	:= 10052;	//Check Limit Error While Overwriting Product
						END_IF

					1:
						tyMagRcpInfoIn	:= p_tyLCSMagRcpInfo;
						eMagRcpAct		:= MagRcpActAddEdit;

						IF (p_eMagRcpStat = MagRcpActAddEdit) AND (p_eMagRcpStatus  = Done) THEN
							eStatus		:= Done;

							IF p_bMagRcpNmEmpty = TRUE THEN
								udiPLCStatus	:= 10053;	//Recipe Name Empty While Overwriting Product
							ELSIF p_bMagRcpListFull = TRUE THEN
								udiPLCStatus	:= 10054;	//Recipe List Full While Overwriting Product
							ELSE
								udiPLCStatus	:= 0;
							END_IF

							eMagRcpAct	:= MagRcpActIdle;

						ELSIF p_eMagRcpStatus = Error THEN
							eStatus			:= Done;
							udiPLCStatus	:= 10055;	//Recipe Program Error While Overwriting Product
						END_IF

				END_CASE

			END_IF
		LCSActDelMag:
			IF eStatus = Idle OR eStatus = Busy THEN

				eStatus			:= Busy;
				udiPLCStatus	:= 65535;

				sStatTxt	:= a_sStatText[eStat];

				CASE usiStep OF
					0:
						bChkMagLmt	:= TRUE;

						IF p_bChkMagLmtOK = TRUE THEN
							usiStep			:= 1;
						ELSIF p_bChkMagLmtNG = TRUE THEN
							eStatus			:= Done;
							udiPLCStatus	:= 10056;	//Check Limit Error While Deleting Product
						END_IF

					1:
						tyMagRcpInfoIn	:= p_tyLCSMagRcpInfo;
						eMagRcpAct	:= MagRcpActDel;

						IF (p_eMagRcpStat = MagRcpActDel) AND (p_eMagRcpStatus = Done) THEN
							eStatus		:= Done;

							IF p_bMagRcpNmEmpty = TRUE THEN
								udiPLCStatus	:= 10057;	//Recipe Name Empty While Deleting Product
							ELSIF p_bProdRcpNmNotExist = TRUE THEN
								udiPLCStatus	:= 10058;	//Recipe Name Not Exist While Deleting Product
							ELSE
								udiPLCStatus	:= 0;
							END_IF

							eMagRcpAct	:= MagRcpActIdle;

						ELSIF p_eMagRcpStatus = Error THEN
							eStatus			:= Done;
							udiPLCStatus	:= 10059;	//Recipe Program Error While Deleting Product
						END_IF

				END_CASE

			END_IF
		LCSActUploadMag:
			IF eStatus = Idle OR eStatus = Busy THEN

				eStatus			:= Busy;
				udiPLCStatus	:= 65535;

				sStatTxt	:= a_sStatText[eStat];

				tyMagRcpInfoIn	:= p_tyLCSMagRcpInfo;
				eMagRcpAct		:= MagRcpActGetInfo;

				IF (p_eMagRcpStat = MagRcpActGetInfo) AND (p_eMagRcpStatus = Done) THEN
					eStatus		:= Done;

					IF p_bMagRcpNmEmpty = TRUE THEN
						udiPLCStatus	:= 10061;	//Magazine Recipe Name Empty While Uploading Product
					ELSIF p_bProdRcpNmNotExist = TRUE THEN
						eStatus			:= Done;
						udiPLCStatus	:= 10061;	//Magazine Recipe Name Not Exist While Uploading Product
					ELSE
						udiPLCStatus		:= 0;
						tyPLCMagRcpInfo	:= p_tyMagRcpInfoOut;
					END_IF

					eMagRcpAct	:= MagRcpActIdle;

				ELSIF p_eMagRcpStatus = Error THEN
					eStatus			:= Done;
					udiPLCStatus	:= 10062;	//Magazine Recipe Program Error While Uploading Product
				END_IF

			END_IF

		ELSE
			IF eStatus = Idle OR eStatus = Busy THEN
				eStatus	:= Done;
			END_IF

	END_CASE

END_ACTION
```

#### Init.st
```iecst
(** 2019-04-24 **)
PROGRAM _INIT

	(* Always Change If Project Change *)

	//Pass Address To Global Address For External Use
	//Action, State & Status
	p_LCSMngRcpStat		:= ADR(eStat);
	p_LCSMngRcpStatus	:= ADR(eStatus);
	p_LCSMngRcpStatTxt	:= ADR(sStatTxt);

	//Alarm
	p_LCSMngRcpAlmData	:= ADR(tyAlmData);

	//Output
	p_LCSMngRcp_PLCStatus		:= ADR(udiPLCStatus);
	p_LCSMngRcp_PLCIdxAct		:= ADR(iPLCIdxAct);
	p_LCSMngRcp_PLCIdxStat		:= ADR(iPLCIdxStat);
	p_LCSMngRcp_PLCProdRcpInfo	:= ADR(tyPLCProdRcpInfo);

	p_LCSMngRcpProdRcpAct		:= ADR(eProdRcpAct);
	p_LCSMngRcpProdRcpInfoIn	:= ADR(tyProdRcpInfoIn);
	p_LCSMngRcpChkLmt			:= ADR(bChkLmt);

	p_LCSMngRcpMagRcpAct		:= ADR(eMagRcpAct);
	p_LCSMngRcpMagRcpInfoIn		:= ADR(tyMagRcpInfoIn);
	p_LCSMngRcp_PLCMagRcpInfo	:= ADR(tyPLCMagRcpInfo);
	p_LCSMngMagRcpChkLmt		:= ADR(bChkMagLmt);
	(* Always Change If Project Change *)

END_PROGRAM
```

### Program Logical/LCS/LCSLF (IEC, version 1.00.0) - 1.00.0 - NtRecipe v5.00.0 , NtFileIO v5.00.0

#### Act_InitGlobal.st - Change By Project
```iecst
(** 2019-05-07 **)
ACTION Act_InitGlobal:

	(* Always Change If Project Change *)

	//Pass Data To Link
	p_bLinkStartupRun ACCESS p_StartupRun;
	p_bLinkNtParamProjLaneBPrep ACCESS p_NtParamProjLaneBPrep;
	p_eLinkMcParamUSACommMod ACCESS p_McParamUSCommAMod;
	p_eLinkMcParamUSBCommMod ACCESS p_McParamUSCommBMod;

	p_bLinkOpsRun ACCESS p_OpsRun;

	//Pass Data To Internal Use
	p_eAct ACCESS p_LCS_LCSLF_LCSAct;
	p_udiRstErr ACCESS p_RstErrReset;
	p_bPrep ACCESS p_NtParamLCSLFPrep;
	p_bEn ACCESS p_McParamLCSLFEn;
	p_tyCurrProdParam ACCESS p_ProdRcpCurrRcp0;
	p_bMnlAccData ACCESS p_McParamMnlAccDat;
	p_bAccData ACCESS p_UIProdAccData;
	p_tyLCSProdRcpInfo ACCESS p_LCS_LCSLF_LCSProdRcpInfo;
	p_bChkLmtOK ACCESS p_LCSChkLmtOK;
	p_bChkLmtNG ACCESS p_LCSChkLmtNG;
	p_sProgNm ACCESS p_NtParamLCSLFProgNm;
	p_bNtSettingsLoadDone ACCESS p_StartupNtSettingsLoadDone;

	//Added
	p_bUIBtnSectionLdr ACCESS p_UISectionLdr;
	p_bLCSSectionLeaderEn ACCESS p_LCSSectionLeaderEn;
	p_bMcParamSectionLdr ACCESS p_McParamSectionLeader;
	p_bLinkConvHvBrd ACCESS p_PshrConvHvBrd;
	(* Always Change If Project Change *)

END_ACTION
```

#### InputRef_Link.var - Change By Project
```iecst
(*2019-04-24*)
(**)
VAR
	sWidthInUMTemp : STRING[80];
	p_bLinkStartupRun : REFERENCE TO BOOL;
END_VAR
(**)
VAR
	p_bLinkNtParamProjLaneBPrep : REFERENCE TO BOOL;
	p_eLinkMcParamUSACommMod : REFERENCE TO eMcSetCommMod;
	p_eLinkMcParamUSBCommMod : REFERENCE TO eMcSetCommMod;
END_VAR
(**)
VAR
	p_bLinkOpsRun : REFERENCE TO BOOL;
	p_bLinkConvHvBrd : REFERENCE TO BOOL;
END_VAR
```

#### Act_LinkEn.st - Change By Project
```iecst
(** 2019-04-24 **)
ACTION Act_LinkEn:

	//Link bPrep, bEn & bDis
	IF p_bLinkNtParamProjLaneBPrep = FALSE THEN
		p_bDis	:= (p_bLinkStartupRun = TRUE) OR (p_eLinkMcParamUSACommMod = McSetCommModHermes);
	ELSE
		p_bDis	:= (p_bLinkStartupRun = TRUE) OR (p_eLinkMcParamUSACommMod = McSetCommModHermes) OR (p_eLinkMcParamUSBCommMod = McSetCommModHermes);
	END_IF

END_ACTION
```

#### Act_Main.st - Do Not Change!!!
```iecst
(** 2019-06-28 **)
ACTION Act_Main:

	//Main
	CASE eStat OF

		LCSActIdle:
			IF eStatus <> Idle THEN	//Reset Data
				//Private
				usiStep		:= 0;
				bAccDataMnl	:= FALSE;
				bChkLmt		:= FALSE;

				tyInfoData.sProgNm		:= '';
				tyInfoData.udiCode		:= 0;
				tyInfoData.eSeverity	:= AlmSeverityNA;
				tyInfoData.sAlmMsg		:= '';

				sStatTxt	:= a_sStatText[eStat];

			END_IF

			eStatus			:= Idle;
			udiPLCStatus	:= 65534;

		LCSActRunProd:
			IF eStatus = Idle OR eStatus = Busy THEN

				eStatus			:= Busy;
				udiPLCStatus	:= 65535;

				sStatTxt	:= a_sStatText[eStat];

				CASE usiStep OF
					0:
						//Check Limit
						bChkLmt	:= TRUE;

						IF p_bChkLmtOK = TRUE THEN
							usiStep			:= 1;
						ELSIF p_bChkLmtNG = TRUE THEN
							eStatus			:= Done;
							udiPLCStatus	:= 10010;	//Out Of Range While Accepting New Recipe
						END_IF

					1:
						//Manual Accept Data Check
						IF p_bMnlAccData = TRUE THEN
							bAccDataMnl	:= TRUE;

							//Info Message
							tyInfoData.sProgNm		:= p_sProgNm;
							tyInfoData.udiCode		:= 10000;
							tyInfoData.eSeverity	:= AlmSeverityInfo;
							tyInfoData.sAlmMsg		:= p_sInfoMsg;

							IF p_bAccData = TRUE THEN
								p_bAccData := FALSE; //2023_07_26_Debug for Manual Accept Data automatically accept after product change many times
								bAccDataMnl	:= FALSE;
								usiStep		:= 2;
							END_IF
						ELSE
							bAccDataMnl	:= FALSE;
							p_bAccData := FALSE; //2023_07_26_Debug for Manual Accept Data automatically accept after product change many times
							usiStep		:= 2;
						END_IF

					2:
						//Accept New Recipe Condition
						IF p_bAccNewRcpCond = TRUE THEN
							usiStep	:= 3;
						ELSE
							//Info Message
							tyInfoData.sProgNm		:= p_sProgNm;
							tyInfoData.udiCode		:= 10000;
							tyInfoData.eSeverity	:= AlmSeverityInfo;
							tyInfoData.sAlmMsg		:= p_sInfoMsg;
						END_IF

					3:
						//Accept New Recipe
						p_tyCurrProdParam	:= p_tyLCSProdRcpInfo;

						IF p_bLCSSectionLeaderEn = TRUE THEN
							p_bMcParamSectionLdr	:= TRUE;
							p_bUIBtnSectionLdr		:= TRUE;
						ELSE
							p_bMcParamSectionLdr	:= FALSE;
							p_bUIBtnSectionLdr		:= FALSE;
						END_IF

						usiStep	:= 4;

					4:
						//Clear Info Message
						tyInfoData.sProgNm		:= '';
						tyInfoData.udiCode		:= 0;
						tyInfoData.eSeverity	:= AlmSeverityNA;
						tyInfoData.sAlmMsg		:= '';

						usiStep	:= 0;

						eStatus			:= Done;
						udiPLCStatus	:= 0;

				END_CASE

			END_IF

		ELSE
			IF eStatus = Idle OR eStatus = Busy THEN
				eStatus	:= Done;
			END_IF

	END_CASE

END_ACTION
```

#### InputRef.var - Do Not Change!!!
```iecst
(*2019-06-28*)
(**)
(*General*)
VAR
	p_eAct : REFERENCE TO eLCSAction;
	p_udiRstErr : REFERENCE TO UDINT;
	p_bPrep : REFERENCE TO BOOL;
	p_bEn : REFERENCE TO BOOL;
	p_bDis : REFERENCE TO BOOL;
END_VAR
(**)
(*Configuration*)
VAR
	p_tyCurrProdParam : REFERENCE TO tyProdRcpParam;
	p_bMnlAccData : REFERENCE TO BOOL;
	p_bAccData : REFERENCE TO BOOL;
	p_tyLCSProdRcpInfo : REFERENCE TO tyProdRcpParam;
	p_bChkLmtOK : REFERENCE TO BOOL;
	p_bChkLmtNG : REFERENCE TO BOOL;
	p_bAccNewRcpCond : REFERENCE TO BOOL;
	p_bUpdtNewRcpCond : REFERENCE TO BOOL;
	p_bAutoUpdtData : REFERENCE TO BOOL;
	p_bUIUpdtData : REFERENCE TO BOOL;
	p_sInfoMsg : REFERENCE TO STRING[200];
	p_sProgNm : REFERENCE TO STRING[15];
	p_bNtSettingsLoadDone : REFERENCE TO BOOL;
END_VAR
(*Section Leader*)
VAR
	p_bUIBtnSectionLdr : REFERENCE TO BOOL;
	p_bLCSSectionLeaderEn : REFERENCE TO BOOL;
	p_bMcParamSectionLdr : REFERENCE TO BOOL;
END_VAR
```

### Ops.var - Change By Project
```iecst
(*2019-04-16*)
(**)
(*Action & State & Status*)
VAR
	p_OpsStat : UDINT;
	p_OpsStatus : UDINT;
	p_OpsStatTxt : UDINT;
END_VAR
(**)
(*Alarm*)
(**)
(*Output*)
VAR
	p_OpsOpsStatus : UDINT;
	p_OpsStatusRun : UDINT;
	p_OpsStatusStop : UDINT;
	p_OpsStatusCycleStop : UDINT;
	p_OpsStatusStep : UDINT;
	p_OpsRun : UDINT;
	p_OpsStop : UDINT;
	p_OpsStep : UDINT;
	p_OpsPause : UDINT;
END_VAR
```

### Program Logical/Operations/Ops (IEC) - 1.00.0 - 

#### InputRef_Link.var
```iecst
(*2019-01-20*)
(**)
(*External*)
VAR
	p_bLinkOpsTravLifULPaused : REFERENCE TO BOOL;
	p_bLinkOpsMagUL1Paused : REFERENCE TO BOOL;
	p_bLinkOpsMagUL2Paused : REFERENCE TO BOOL;
	p_bLinkOpsMagUL3Paused : REFERENCE TO BOOL;
	p_bLinkOpsMagConvUL1Paused : REFERENCE TO BOOL;
	p_bLinkOpsMagConvUL2Paused : REFERENCE TO BOOL;
	p_bLinkOpsMagConvUL3Paused : REFERENCE TO BOOL;
	p_bLinkOpsInMagConvPaused : REFERENCE TO BOOL;
	p_bLinkOpsOutMagConvPaused : REFERENCE TO BOOL;
	p_bLinkOpsMagConvStprPaused : REFERENCE TO BOOL;
	p_bLinkOpsMagConv2StprPaused : REFERENCE TO BOOL;
	p_bLinkUIOpsAct : REFERENCE TO eOperationsAction;
	p_bLinkSimuRun : REFERENCE TO BOOL;
	p_bLinkSimuStop : REFERENCE TO BOOL;
	p_bLinkOpsLifMagULPaused : REFERENCE TO BOOL;
	p_bLinkProjLifterMagPlatform : REFERENCE TO BOOL;
	p_bLinkProjMagConvLanePrep : REFERENCE TO BOOL;
END_VAR
```

#### Act_InitGlobal.st
```iecst
(** 2019-03-22 **)
ACTION Act_InitGlobal:

	(* Always Change If Project Change *)

	//Pass Data To Link
	p_bLinkOpsTravLifULPaused ACCESS p_OpsTravLifULPaused;
//	p_bLinkOpsMagUL1Paused ACCESS p_OpsMagUL1Paused;
//	p_bLinkOpsMagUL2Paused ACCESS p_OpsMagUL2Paused;
//	p_bLinkOpsMagUL3Paused ACCESS p_OpsMagUL3Paused;
	p_bLinkOpsMagConvUL1Paused ACCESS p_OpsMagConvUL1Paused;
	p_bLinkOpsMagConvUL2Paused ACCESS p_OpsMagConvUL2Paused;
	p_bLinkOpsMagConvUL3Paused ACCESS p_OpsMagConvUL3Paused;
	p_bLinkOpsLifMagULPaused ACCESS p_OpsLifMagULPaused;
	p_bLinkOpsInMagConvPaused ACCESS p_OpsInMagConvPaused;
	p_bLinkOpsOutMagConvPaused ACCESS p_OpsOutMagConvPaused;
	p_bLinkOpsMagConvStprPaused ACCESS p_OpsMagConvStprPaused;
	p_bLinkOpsMagConv2StprPaused ACCESS p_OpsMagConv2StprPaused;

	p_bLinkProjLifterMagPlatform ACCESS p_NtParamProjLifterMagPlatform;
	p_bLinkProjMagConvLanePrep ACCESS p_NtParamProjMagConvLane1Prep;

	p_bLinkUIOpsAct ACCESS p_UIOpsAct;
	p_bLinkSimuRun ACCESS p_SimuRun;
	p_bLinkSimuStop ACCESS p_SimuStop;
	//Pass Data To Internal Use
//	p_eAct ACCESS p_UIOpsAct;
	p_udiRstErr ACCESS p_RstErrReset;
	p_bNtSettingsLoadDone ACCESS p_StartupNtSettingsLoadDone;

	(* Always Change If Project Change *)

END_ACTION
```

#### Act_Link.st
```iecst
(** 2019-01-20 **)
ACTION Act_Link:

	IF p_bLinkProjLifterMagPlatform AND NOT(p_bLinkProjMagConvLanePrep) THEN
		p_bPaused	:= p_bLinkOpsTravLifULPaused AND p_bLinkOpsLifMagULPaused;
	ELSIF p_bLinkProjMagConvLanePrep THEN
		p_bPaused	:=  p_bLinkOpsLifMagULPaused AND p_bLinkOpsInMagConvPaused AND p_bLinkOpsOutMagConvPaused AND p_bLinkOpsMagConvStprPaused
						AND p_bLinkOpsMagConv2StprPaused;
	ELSE

		p_bPaused	:= p_bLinkOpsTravLifULPaused
					(*AND p_bLinkOpsMagUL1Paused AND p_bLinkOpsMagUL2Paused AND p_bLinkOpsMagUL3Paused*)
						AND p_bLinkOpsMagConvUL1Paused AND p_bLinkOpsMagConvUL2Paused AND p_bLinkOpsMagConvUL3Paused;

	END_IF

END_ACTION
```

#### Act_LinkAction.st
```iecst
(** 2019-03-29 **)
ACTION Act_LinkAction:

	IF p_bLinkUIOpsAct <> OperationsActIdle THEN
		p_eAct ACCESS p_UIOpsAct;
	ELSIF EDGEPOS(p_bLinkSimuRun) THEN
		p_eAct := OperationsActStart;
	ELSIF EDGEPOS(p_bLinkSimuStop) THEN
		p_eAct := OperationsActStop;
	END_IF

	IF (eStat = OperationsActStart OR eStat = OperationsActStop) AND  eStatus = Done THEN
		eAct := OperationsActIdle;
		p_eAct := OperationsActIdle;
	END_IF

END_ACTION
```

#### Init.st
```iecst
(** 2019-04-16 **)
PROGRAM _INIT

	(* Always Change If Project Change *)

	//Pass Address To Global Address For External Use
	//Action, State & Status
	p_OpsStat		:= ADR(eStat);
	p_OpsStatus		:= ADR(eStatus);
	p_OpsStatTxt	:= ADR(sStatTxt);

	//Alarm

	//Output
	p_OpsOpsStatus			:= ADR(eOpsStatus);
	p_OpsStatusRun			:= ADR(bStatusRun);
	p_OpsStatusStop			:= ADR(bStatusStop);
	p_OpsStatusCycleStop	:= ADR(bStatusCycleStop);
	p_OpsStatusStep			:= ADR(bStatusStep);
	p_OpsRun				:= ADR(bRun);
	p_OpsStop				:= ADR(bStop);
	p_OpsStep				:= ADR(bStep);
	p_OpsPause				:= ADR(bPaused);
	(* Always Change If Project Change *)

END_PROGRAM
```

### OpsTravLifUL.typ - Do Not Change!!!
```iecst
(*2018-12-11*)
(**)
(*Configuration*)

TYPE
	eULMod :
		(
		ULModUnloadFrontLnA,
		ULModRejFrontLnA,
		ULModRejFrontLnARev,
		ULModUnloadRearLnB,
		ULModRejRearLnB,
		ULModRejRearLnBRev,
		ULModUnloadDualLnAB,
		ULModRejDualLnA,
		ULModRejDualLnB
		);
	eULMag :
		(
		ULMagDual,
		ULMagTriple,
		ULMagQuadruple
		);
END_TYPE

(**)

TYPE
	tyParamTravLifUL : 	STRUCT
		a_bUSDis : ARRAY[1..3]OF BOOL := [3(FALSE)];
		a_bDSDis : ARRAY[1..3]OF BOOL := [3(FALSE)];
		a_usiUSPriority : ARRAY[1..3]OF USINT := [1,2,3];
		a_usiDSPriority : ARRAY[1..3]OF USINT := [1,2,3];
		a_bMagRej : ARRAY[1..3]OF BOOL := [3(FALSE)];
	END_STRUCT;
END_TYPE

(**)
(*Sequence*)

TYPE
	eTravLifULStep :
		(
		TravLifULStepNA,
		TravLifULStepInitConv,
		TravLifULStepInitInletPneuCls,
		TravLifULStepInitInOutPneuCls,
		TravLifULStepInitTravLif,
		TravLifULStepInitAWTravLif,
		TravLifULStepAWMov,
		TravLifULStepScanDS,
		TravLifULStepHermesBCode,
		TravLifULStepWaitReturnCode,
		TravLifULStepMagChkReturnCode,
		TravLifULStepTravLifMov,
		TravLifULStepUSSigWait,
		TravLifULStepUSSigRechk,
		TravLifULStepInletPneuOpn,
		TravLifULStepUSSigRechkTwice,
		TravLifULStepUSMagWidthChk,
		TravLifULStepStopperRet,
		TravLifULStepUSComm,
		TravLifULStepEntBrd,
		TravLifULStepInletPneuCls,
		TravLifULStepStopperExt,
		TravLifULStepDSSigWait,
		TravLifULStepDSSigRechk,
		TravLifULStepOutletPneuOpn,
		TravLifULStepDSSigRechkTwice,
		TravLifULStepDSMagWidthChk,
		TravLifULStepDSComm,
		TravLifULStepExitBrd,
		TravLifULStepOutletPneuCls,
		TravLifULStepScanStdBy,
		TravLifULStepTranOutErr,
		TravULStepTranOutBrdStuckErr,
		TravULStepTranInBrdStuckErr,
		TravULStepClrSensorErr,
		TravLifULStepMagWidthErr,
		TravULStepBrdLostInMiddle,
		TravULStepClrSensorErrBefTrav
		);
	eTravLifULPos :
		(
		TravLifULPosInvalid,
		TravLifULPosUS1,
		TravLifULPosUS2,
		TravLifULPosUS3,
		TravLifULPosDS1,
		TravLifULPosDS2,
		TravLifULPosDS3
		);
	tyMagCoord : 	STRUCT
		usiMagPos : USINT;
		usiMagSlot : USINT;
	END_STRUCT;
END_TYPE
```

### OpsTravLifUL.var - Change By Project
```iecst
(*2019-03-25*)
(**)
(*Action & State & Status*)
(**)
(*Alarm*)
VAR
	p_OpsTravLifULAlmData : UDINT;
END_VAR
(**)
(*Output*)
VAR
	p_OpsTravLifULStepTxt : UDINT;
	p_OpsTravLifULPaused : UDINT;
END_VAR
(**)
VAR
	p_OpsTravLifULUSSMEMAAct1 : UDINT;
	p_OpsTravLifULUSSMEMAAct2 : UDINT;
	p_OpsTravLifULUSSMEMAAct3 : UDINT;
	p_OpsTravLifULDSSMEMAAct1 : UDINT;
	p_OpsTravLifULDSSMEMAAct2 : UDINT;
	p_OpsTravLifULDSSMEMAAct3 : UDINT;
	p_OpsTravLifULConvAct : UDINT;
	p_OpsTravLifULAWPushPullAct : UDINT;
	p_OpsTravLifULAWAct : UDINT;
	p_OpsTravLifULTravAct : UDINT;
	p_OpsTravLifULLifAct : UDINT;
	p_OpsTravLifULInletPneuAct : UDINT;
	p_OpsTravLifULOutletPneuAct : UDINT;
	p_OpsTravLifULOutletPneuAct2 : UDINT;
	p_OpsTravLifULOutletPneuAct3 : UDINT;
	p_OpsTravLifULStopperAct1 : UDINT;
	p_OpsTravLifULStopperAct2 : UDINT;
	p_OpsTravLifULStopperAct3 : UDINT;
END_VAR
(**)
VAR
	p_OpsTravLifULPosGo : UDINT;
	p_OpsTravLifULMagDis : UDINT;
	p_OpsTravLifULMagRej : UDINT;
	p_OpsTravLifULInitConv : UDINT;
	p_OpsTravLifULInitDone : UDINT;
	p_OpsTravLifULUSComm : UDINT;
	p_OpsTravLifULEntBrd : UDINT;
	p_OpsTravLifULDSComm : UDINT;
	p_OpsTravLifULExitBrd : UDINT;
	p_OpsTravLifULTravLifMov : UDINT;
	p_OpsTravLifULSelfTest : UDINT;
	p_OpsTravLifULTravGotoChkPt : UDINT;
	p_OpsTravLifULInDSPos : UDINT;
	p_OpsTravLifULUSWidthChkBrdExist : UDINT;
	p_OpsTravLifULJogSpeed : UDINT;
	p_OpsTravLifULStpExt : UDINT;
	p_OpsTravLifULBypCurtainSenCtrl : UDINT;
	p_OpsTravLifULBypCurtainLED : UDINT;
	p_OpsTravLifULMagWidthChk : UDINT;
	p_OpsTravLifULMagWidthChkStep : UDINT;
	p_OpsTravLifULTopScan : UDINT;
	p_OpsTravLifULBtmScan : UDINT;
	p_OpsTravLifULBarcode : UDINT;
	p_OpsTravLifULMsgReq : UDINT;
	p_OpsTravLifWChkErrCmdUnclmp1 : UDINT;
	p_OpsTravLifWChkErrCmdUnclmp2 : UDINT;
	p_OpsTravLifWChkErrCmdUnclmp3 : UDINT;
	p_OpsTravLifParamTravLif : UDINT;
	p_OpsTravLifOpsModGonethrough : UDINT;
	p_OpsTravLifWGdBrdChk : UDINT;
	p_OpsTravLifAllwExitMag1 : UDINT;
	p_OpsTravLifAllwExitMag2 : UDINT;
	p_OpsTravLifAllwExitMag3 : UDINT;
	p_OpsTravLifULPartProcessItms : UDINT;
	p_OpsTravLifULMagEntered : UDINT;
	p_OpsTravLifInletStprAct : UDINT;
	p_OpsTravLifStartScanSig : UDINT;
	p_OpsTravLifMag1TransOut : UDINT;
	p_OpsTravLifMag2TransOut : UDINT;
	p_OpsTravLifMag3TransOut : UDINT;
	p_OpsTravLifOpsStep : UDINT;
	p_OpsTravLifGotoOpsStep : UDINT;
	p_OpsTravLifScanCntr : UDINT;
END_VAR
```

### Program Logical/Operations/OpsTravLifUL (IEC, version 1.00.0) - 1.00.0 - 

#### Init.st - Change By Project
```iecst
(** 2019-03-25 **)
PROGRAM _INIT

	(* Always Change If Project Change *)

	//Pass Address To Global Address For External Use
	//Action, State & Status

	//Alarm
	p_OpsTravLifULAlmData	:= ADR(tyAlmData);

	//Output
	p_OpsTravLifULStepTxt			:= ADR(sStepTxt);
	p_OpsTravLifULPaused			:= ADR(bPaused);

	p_OpsTravLifULUSSMEMAAct1		:= ADR(eUSSMEMAAct1);
	p_OpsTravLifULUSSMEMAAct2 		:= ADR(eUSSMEMAAct2);
	p_OpsTravLifULUSSMEMAAct3		:= ADR(eUSSMEMAAct3);
	p_OpsTravLifULDSSMEMAAct1		:= ADR(eDSSMEMAAct1);
	p_OpsTravLifULDSSMEMAAct2		:= ADR(eDSSMEMAAct2);
	p_OpsTravLifULDSSMEMAAct3		:= ADR(eDSSMEMAAct3);
	p_OpsTravLifULConvAct			:= ADR(eConvAct);
	p_OpsTravLifULAWAct				:= ADR(eAWAct);
	p_OpsTravLifULAWPushPullAct		:= ADR(eAWPushOrPullerAct);
	p_OpsTravLifULTravAct			:= ADR(eTravAct);
	p_OpsTravLifULLifAct			:= ADR(eLifAct);
	p_OpsTravLifULInletPneuAct		:= ADR(eInletPneuAct);
	p_OpsTravLifULOutletPneuAct		:= ADR(eOutletPneuAct);
	p_OpsTravLifULOutletPneuAct2	:= ADR(eOutletPneuAct2);
	p_OpsTravLifULOutletPneuAct3	:= ADR(eOutletPneuAct3);
	p_OpsTravLifULStopperAct1		:= ADR(eStopperAct1);
	p_OpsTravLifULStopperAct2		:= ADR(eStopperAct2);
	p_OpsTravLifULStopperAct3		:= ADR(eStopperAct3);

	p_OpsTravLifULPosGo				:= ADR(eTravLifPosGo);
	p_OpsTravLifULMagDis			:= ADR(a_bMagDis);
	p_OpsTravLifULMagRej			:= ADR(a_bMagRej);
	p_OpsTravLifULInitConv			:= ADR(bInitConv);
	p_OpsTravLifULInitDone			:= ADR(bOpsInitDone);
	p_OpsTravLifULUSComm			:= ADR(bUSComm);
	p_OpsTravLifULEntBrd			:= ADR(bEntBrd);
	p_OpsTravLifULDSComm			:= ADR(bDSComm);
	p_OpsTravLifULExitBrd			:= ADR(bExitBrd);
	p_OpsTravLifULTravLifMov		 := ADR(bTravLifMove);
	p_OpsTravLifULUSWidthChkBrdExist	:= ADR(bUSWidthChkBrdExist);
	p_OpsTravLifULStpExt				:= ADR(bStopperExtStep);

	p_OpsTravLifULJogSpeed				:= ADR(udiJogSpeed);

	p_OpsTravLifULSelfTest				:= ADR(bSelfTest);
	p_OpsTravLifULInDSPos				:= ADR(bTravLifInDSPos);

	p_OpsTravLifULBypCurtainLED 		:= ADR (bBypCurtainSensorPBLED);
	p_OpsTravLifULBypCurtainSenCtrl		:= ADR (bBypCurtainSenCtrl);

	p_OpsTravLifULTravGotoChkPt			:= ADR (bTravGoToChkPt);
	p_OpsTravLifULMagWidthChk	 		:= ADR(bMagWidthChk);
	p_OpsTravLifULMagWidthChkStep 		:= ADR(usiMagWidthChkStep);

	p_OpsTravLifULTopScan			:= ADR(eTCPTopAct);
	p_OpsTravLifULBtmScan			:= ADR(eTCPBtmAct);
	p_OpsTravLifULBarcode				:= ADR(sBarcode);
	p_OpsTravLifULMsgReq				:= ADR(tyOpConMsgReq);
	p_OpsTravLifULPartProcessItms := ADR(tyPartProcessedItems);
	p_OpsTravLifULMagEntered 			:= ADR(asMagEntered);

	p_OpsTravLifWChkErrCmdUnclmp1		:= ADR (bWidthChkErrCmdUnclmp1); //To OpsMagConvUL 1,2,3
	p_OpsTravLifWChkErrCmdUnclmp2		:= ADR (bWidthChkErrCmdUnclmp2);
	p_OpsTravLifWChkErrCmdUnclmp3		:= ADR (bWidthChkErrCmdUnclmp3);

	p_OpsTravLifParamTravLif			:= ADR(tyParamTravLif); //seperate calculation for US and DS

	p_OpsTravLifOpsModGonethrough   := ADR(bOpsModGonethrough);

	p_OpsTravLifWGdBrdChk  := ADR(bGdChk);
	p_OpsTravLifAllwExitMag1 	:= ADR(bAllwExitMag1);
	p_OpsTravLifAllwExitMag2	:= ADR(bAllwExitMag2);
	p_OpsTravLifAllwExitMag3	:= ADR(bAllwExitMag3);

	//inlet stopper
	p_OpsTravLifInletStprAct	:= ADR(eInletStopperAct);

	//OpsScanner
	p_OpsTravLifStartScanSig := ADR(bStartScanSig);
	p_OpsTravLifMag1TransOut := ADR(bPCBExitMag1);
	p_OpsTravLifMag2TransOut := ADR(bPCBExitMag2);
	p_OpsTravLifMag3TransOut := ADR(bPCBExitMag3);

	//check eops
	p_OpsTravLifOpsStep := ADR(eOpsStep);
	p_OpsTravLifGotoOpsStep := ADR(eGotoOpsStep);

	//scanner
	p_OpsTravLifScanCntr := ADR(usiScanCntr);
	(* Always Change If Project Change *)

END_PROGRAM
```
